FUNCTION_BLOCK "AutoSusDoor"	// FB 20
TITLE = pneum.RüstplTüren
//------------------------------------------------------------------------------
//version:      0.1 / 10.09.2007
//author:       H.Scheuenstuhl
//modification: Prototyp
//------------------------------------------------------------------------------
AUTHOR : SPAC_slh
FAMILY : AUTOMAT
NAME : SusDoor
VERSION : 0.1
VAR_INPUT
  iMode : BYTE ;	//Funktion:
  iSafetyEdgeMonitoringTim : BYTE ;	//Zeit Schaltleistenüberwachung (in 0.1 sek, BCD-codiert!)
  iOnly1SusDoor : BOOL ;	//einflügelige Rüstplatztür (links)
  iAutoReverse : BOOL ;	//0: sofort.Abschalten  1: Reversierbetrieb wenn Schaltleiste betätigt
END_VAR
VAR
  fk : ARRAY  [0 .. 15 ] OF //Flankenhilfsmerker [n]
  BOOL ;
  hvFEin : BOOL ;	//Hauptventil Fehler:Einschaltüberwachung
  hvFUnt : BOOL ;	//Hauptventil Fehler:Unterbrechungsüberwachung
  LBewTzu : BOOL ;	//letzte Bewegung:Türen schliessen
  SafetyEdgeActuated : BOOL ;	//Schaltleiste betätigt (wenn Türe(n) nicht geschlossen)
  SafetyEdgeReverseMove : BOOL ;	//Schaltleiste betätigt: Türen Rücklauf = Öffnen (Reversierung)
  SafetyEdgePressureOff : BOOL ;	//Schaltleiste betätigt: Pneumatik Druck aus
  SfCloseDoor : BOOL ;	//Schritt fertig:Tür schliessen
  SfOpenDoor : BOOL ;	//Schritt fertig:Tür öffnen
  oeffnFEin : BOOL ;	//Drucküberwachung RpTüren öffnen Fehler:Einschaltüberwachung
  oeffnFUnt : BOOL ;	//Drucküberwachung RpTüren öffnen Fehler:Unterbrechungsüberwachung
  schlFEin : BOOL ;	//Drucküberwachung RpTüren schliessen Fehler:Einschaltüberwachung
  schlFUnt : BOOL ;	//Drucküberwachung RpTüren schliessen Fehler:Unterbrechungsüberwachung
  Luftvh : BOOL ;	//Druckluft für Antrieb der Rüstplatztüren vorhanden
  LockManualOperate : BOOL ;	//Tastensperre nach Fehlbedienung
  SrCloseDoor : BOOL ;	//Schritt:Türen schliessen
  SrOpenDoor : BOOL ;	//Schritt:Türen öffnen
END_VAR
VAR_TEMP
  svAr1 : DWORD ;
  WertInt : INT ;	//Wert integer
  SLUeZeit : S5TIME ;	//s5-Zeitwert Schaltleistenüberwachung
  Mod : ARRAY  [0 .. 15 ] OF //Modus dekodiert, 1 aus 16
  BOOL ;
  LOp0 : BOOL ;	//lokaler Operationsmerker 0, Zwischenmerker
  LOp1 : BOOL ;	//lokaler Operationsmerker 1, Zwischenmerker
  Fa : BOOL ;	//Freigabe Ausgänge
  SusDoorAutoOpen : BOOL ;	//Modus: Rüstplatztür automatisch öffnen nach Palettenwechsel
  AutoEnablePc : BOOL ;	//Modus:automatisches Setzen der PW-Freigabe nach Rüstplatztür zu
  SusDoorOpened : BOOL ;	//Rüstlatztüren sind vollständig geöffnet
  ModeSusDoorAdjust : BOOL ;	//Rüstplatztüren: Betriebsart Einrichten
  ModeSusDoorAuto : BOOL ;	//Rüstplatztüren: Betriebsart Automatik
  AnfTzu1 : BOOL ;	//Anforderung Türen schliessen
  AnfTauf1 : BOOL ;	//Anforderung Türen öffnen
  MachineOn : BOOL ;	//Maschine ist ein
  afbTzu : BOOL ;	//Türen schliessen ausführbar
  afbTauf : BOOL ;	//Türen öffnen ausführbar
  SusDoorFault : BOOL ;	//Sammelsignal: Rüstplatztür(en) gestört
  CloseManual : BOOL ;	//Taster: Türen schliessen
  OpenManual : BOOL ;	//Taster: Türen öffnen
  CloseByRobot : BOOL ;	//Werkstücklader: Türen schliessen
  OpenByRobot : BOOL ;	//Werkstücklader: Türen öffnen
END_VAR
BEGIN
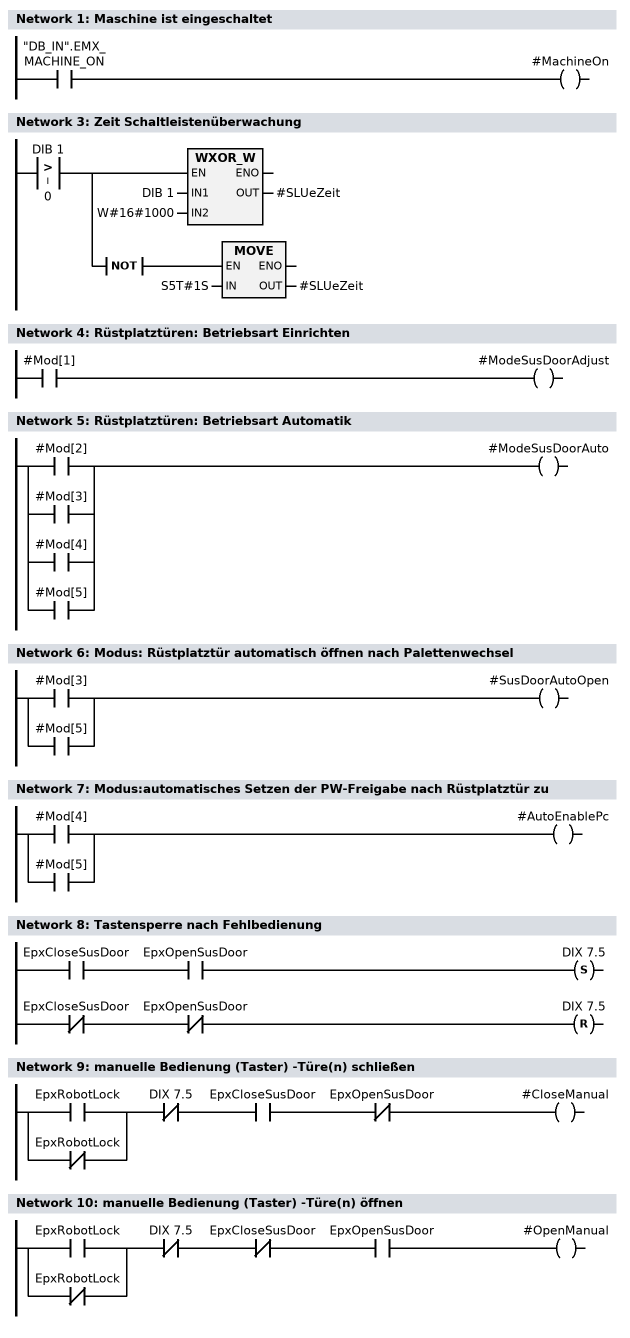
NETWORK
TITLE = Maschine ist eingeschaltet
      A     "DB_IN".EMX_MACHINE_ON;
      =     #MachineOn;
NETWORK
TITLE = iModus dekodieren
//Modus_1: Handbetrieb, Einrichtbetrieb, Tippbetrieb
//Modus_2: Tippen fährt bis Endlage erreicht
//Modus_3: Tippen fährt bis Endlage erreicht
//         nach PW fährt Türe automatisch auf
//Modus_4: Tippen fährt bis Endlage erreicht
//         nach Schließen wird PW-Freigabe gesetzt
//Modus_5: Tippen fährt bis Endlage erreicht
//         nach PW fährt Türe automatisch auf
//         nach Schließen wird PW-Freigabe gesetzt
      L     DIB 0;
      AW    W#16#F;	//Begrenzung auf 0..15, dadurch keine weitere Prüfung erforderlich
      TAR1  #svAr1;
      LAR1  P##Mod;
      L     B#16#0;
      T     LW [AR1,P#0.0];
      TAK;
      +AR1;
      A     "M_HIGH";
      S     L [AR1,P#0.0];
      LAR1  #svAr1;
NETWORK
TITLE = Zeit Schaltleistenüberwachung
//Zuordnung der Zeit (über Konstante S5T); Dekadenbyte = 1 ==> 0,1sec
      L     DIB 1;
      L     0;
      >I;
      =     L 13.0;
      A     L 13.0;
      JNB   _001;
      L     DIB 1;
      L     W#16#1000;
      XOW;
      T     #SLUeZeit;
_001: NOP   0;
      A     L 13.0;
      NOT;
      JNB   _002;
      L     S5T#1S;
      T     #SLUeZeit;
_002: NOP   0;
NETWORK
TITLE = Rüstplatztüren: Betriebsart Einrichten
//Modus_1: Handbetrieb, Einrichtbetrieb, Tippbetrieb
      A     #Mod[1];
      =     #ModeSusDoorAdjust;
NETWORK
TITLE = Rüstplatztüren: Betriebsart Automatik
//Modus_2: Tippen fährt bis Endlage erreicht
//Modus_3: Tippen fährt bis Endlage erreicht
//         nach PW fährt Türe automatisch auf
//Modus_4: Tippen fährt bis Endlage erreicht
//         nach Schließen wird PW-Freigabe gesetzt
//Modus_5: Tippen fährt bis Endlage erreicht
//         nach PW fährt Türe automatisch auf
//         nach Schließen wird PW-Freigabe gesetzt
      O     #Mod[2];
      O     #Mod[3];
      O     #Mod[4];
      O     #Mod[5];
      =     #ModeSusDoorAuto;
NETWORK
TITLE = Modus: Rüstplatztür automatisch öffnen nach Palettenwechsel
//Modus_3: Tippen fährt bis Endlage erreicht
//         nach PW fährt Türe automatisch auf
//Modus_5: Tippen fährt bis Endlage erreicht
//         nach PW fährt Türe automatisch auf
//         nach Schließen wird PW-Freigabe gesetzt
      O     #Mod[3];
      O     #Mod[5];
      =     #SusDoorAutoOpen;
NETWORK
TITLE = Modus:automatisches Setzen der PW-Freigabe nach Rüstplatztür zu
//Modus_4: Tippen fährt bis Endlage erreicht
//         nach Schließen wird PW-Freigabe gesetzt
//Modus_5: Tippen fährt bis Endlage erreicht
//         nach PW fährt Türe automatisch auf
//         nach Schließen wird PW-Freigabe gesetzt
      O     #Mod[4];
      O     #Mod[5];
      =     #AutoEnablePc;
NETWORK
TITLE = Tastensperre nach Fehlbedienung
      A     "EpxCloseSusDoor";
      A     "EpxOpenSusDoor";
      S     DIX 7.5;
      AN    "EpxCloseSusDoor";
      AN    "EpxOpenSusDoor";
      R     DIX 7.5;
      NOP   0;
NETWORK
TITLE = manuelle Bedienung (Taster) -Türe(n) schließen
      A(;
      O     "EpxRobotLock";
      ON    "EpxRobotLock";
      );
      AN    DIX 7.5;
      A     "EpxCloseSusDoor";
      AN    "EpxOpenSusDoor";
      =     #CloseManual;
NETWORK
TITLE = manuelle Bedienung (Taster) -Türe(n) öffnen
      A(;
      O     "EpxRobotLock";
      ON    "EpxRobotLock";
      );
      AN    DIX 7.5;
      AN    "EpxCloseSusDoor";
      A     "EpxOpenSusDoor";
      =     #OpenManual;
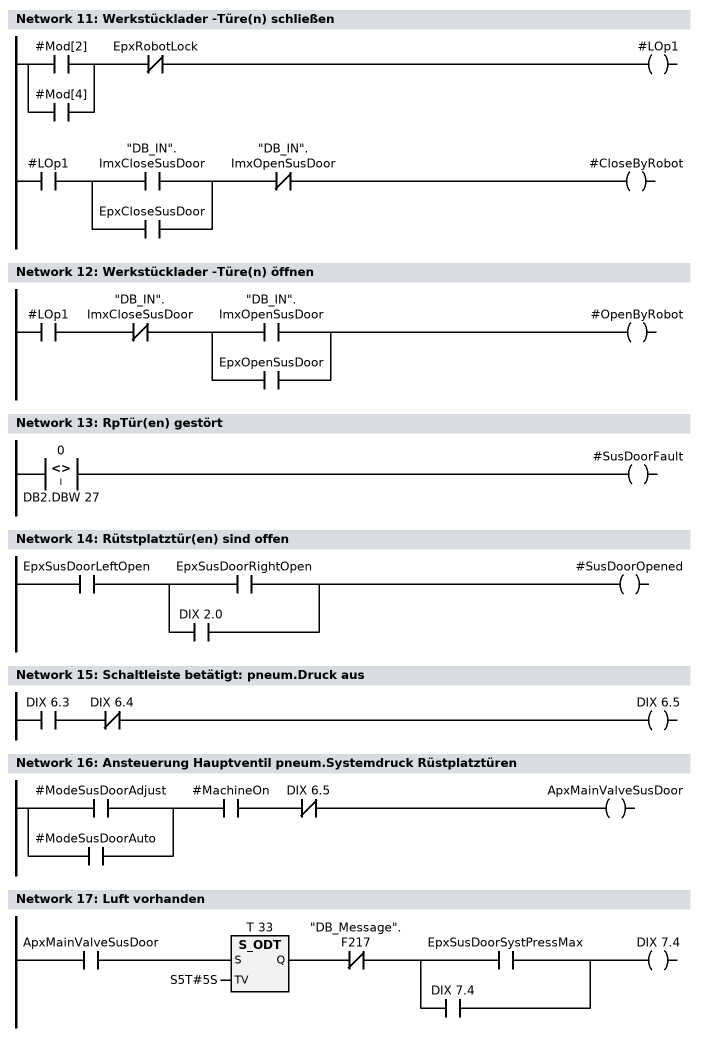
NETWORK
TITLE = Werkstücklader -Türe(n) schließen
//Modus_2: Tippen fährt bis Endlage erreicht
//Modus_4: Tippen fährt bis Endlage erreicht
//         nach Schließen wird PW-Freigabe gesetzt
      A(;
      O     #Mod[2];
      O     #Mod[4];
      );
      AN    "EpxRobotLock";
      =     #LOp1;
      A     #LOp1;
      A(;
      O     "DB_IN".ImxCloseSusDoor;
      O     "EpxCloseSusDoor";
      );
      AN    "DB_IN".ImxOpenSusDoor;
      =     #CloseByRobot;
NETWORK
TITLE = Werkstücklader -Türe(n) öffnen
      A     #LOp1;
      AN    "DB_IN".ImxCloseSusDoor;
      A(;
      O     "DB_IN".ImxOpenSusDoor;
      O     "EpxOpenSusDoor";
      );
      =     #OpenByRobot;
NETWORK
TITLE = RpTür(en) gestört
//DB2.DBW27 = Fehlermeldungen 217 bis 232
      L     0;
      L     DB2.DBW 27;
      <>I;
      =     #SusDoorFault;
NETWORK
TITLE = Rütstplatztür(en) sind offen
//Wenn nur eine Rüstplatztüre ausgewählt wird, dann ist die "rechte Türe" 
//gebrückt.
      A     "EpxSusDoorLeftOpen";
      A(;
      O     "EpxSusDoorRightOpen";
      O     DIX 2.0;
      );
      =     #SusDoorOpened;
NETWORK
TITLE = Schaltleiste betätigt: pneum.Druck aus
      A     DIX 6.3;
      AN    DIX 6.4;
      =     DIX 6.5;
NETWORK
TITLE = Ansteuerung Hauptventil pneum.Systemdruck Rüstplatztüren
      A(;
      O     #ModeSusDoorAdjust;
      O     #ModeSusDoorAuto;
      );
      A     #MachineOn;
      AN    DIX 6.5;
      =     "ApxMainValveSusDoor";
NETWORK
TITLE = Luft vorhanden
      A(;
      A     "ApxMainValveSusDoor";
      L     S5T#5S;
      SD    T 33;
      NOP   0;
      NOP   0;
      NOP   0;
      A     T 33;
      );
      AN    "DB_Message".F217;
      A(;
      O     "EpxSusDoorSystPressMax";
      O     DIX 7.4;
      );
      =     DIX 7.4;
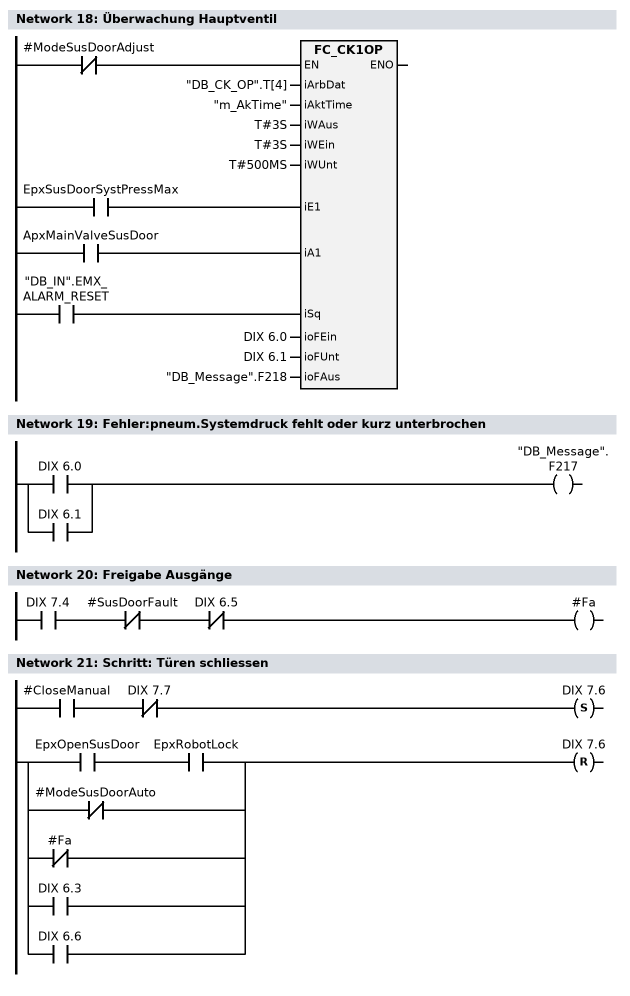
NETWORK
TITLE = Überwachung Hauptventil
      A     "EpxSusDoorSystPressMax";
      =     L 13.0;
      BLD   103;
      A     "ApxMainValveSusDoor";
      =     L 13.1;
      BLD   103;
      A     "DB_IN".EMX_ALARM_RESET;
      =     L 13.2;
      BLD   103;
      AN    #ModeSusDoorAdjust;
      JNB   _003;
      CALL  "FC_CK1OP" (
           iArbDat                  := "DB_CK_OP".T[4],
           iAktTime                 := "m_AkTime",
           iWAus                    := T#3S,
           iWEin                    := T#3S,
           iWUnt                    := T#500MS,
           iE1                      := L 13.0,
           iA1                      := L 13.1,
           iSq                      := L 13.2,
           ioFEin                   := DIX 6.0,
           ioFUnt                   := DIX 6.1,
           ioFAus                   := "DB_Message".F218);
_003: NOP   0;
NETWORK
TITLE = Fehler:pneum.Systemdruck fehlt oder kurz unterbrochen
      O     DIX 6.0;
      O     DIX 6.1;
      =     "DB_Message".F217;
NETWORK
TITLE = Freigabe Ausgänge
      A     DIX 7.4;
      AN    #SusDoorFault;
      AN    DIX 6.5;
      =     #Fa;
NETWORK
TITLE = Schritt: Türen schliessen
      A     #CloseManual;
      AN    DIX 7.7;
      S     DIX 7.6;
      A(;
      A     "EpxOpenSusDoor";
      A     "EpxRobotLock";
      ON    #ModeSusDoorAuto;
      ON    #Fa;
      O     DIX 6.3;
      O     DIX 6.6;
      );
      R     DIX 7.6;
      NOP   0;
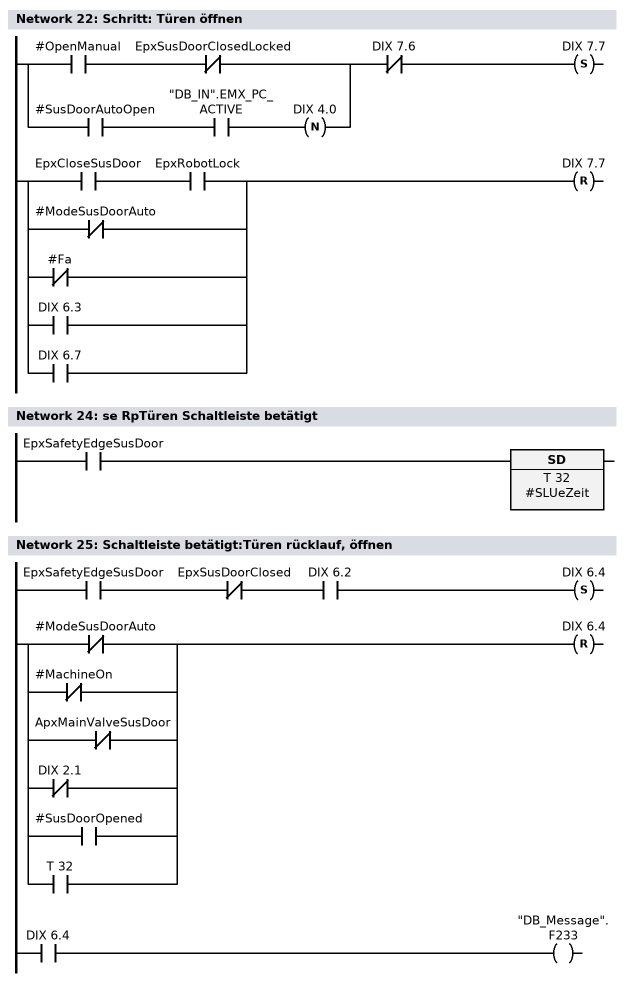
NETWORK
TITLE = Schritt: Türen öffnen
      A(;
      A     #OpenManual;
      AN    "EpxSusDoorClosedLocked";
      O(;
      A     #SusDoorAutoOpen;
      A     "DB_IN".EMX_PC_ACTIVE;
      FN    DIX 4.0;
      );
      );
      AN    DIX 7.6;
      S     DIX 7.7;
      A(;
      A     "EpxCloseSusDoor";
      A     "EpxRobotLock";
      ON    #ModeSusDoorAuto;
      ON    #Fa;
      O     DIX 6.3;
      O     DIX 6.7;
      );
      R     DIX 7.7;
      NOP   0;
NETWORK
TITLE = Schaltleiste an Rüstplatztüren betätigt
      A(;
      A     "DB_IN".EMX_ALARM_RESET;
      R     DIX 6.3;
      A     "EpxSafetyEdgeSusDoor";
      AN    "EpxSusDoorClosed";
      S     DIX 6.3;
      A     DIX 6.3;
      );
      AN    "DB_Message".F233;
      =     "DB_Message".F234;
NETWORK
TITLE = se RpTüren Schaltleiste betätigt
      A     "EpxSafetyEdgeSusDoor";
      L     #SLUeZeit;
      SD    T 32;
NETWORK
TITLE = Schaltleiste betätigt:Türen rücklauf, öffnen
      A     "EpxSafetyEdgeSusDoor";
      AN    "EpxSusDoorClosed";
      A     DIX 6.2;
      S     DIX 6.4;
      A(;
      ON    #ModeSusDoorAuto;
      ON    #MachineOn;
      ON    "ApxMainValveSusDoor";
      ON    DIX 2.1;
      O     #SusDoorOpened;
      O     T 32;
      );
      R     DIX 6.4;
      A     DIX 6.4;
      =     "DB_Message".F233;
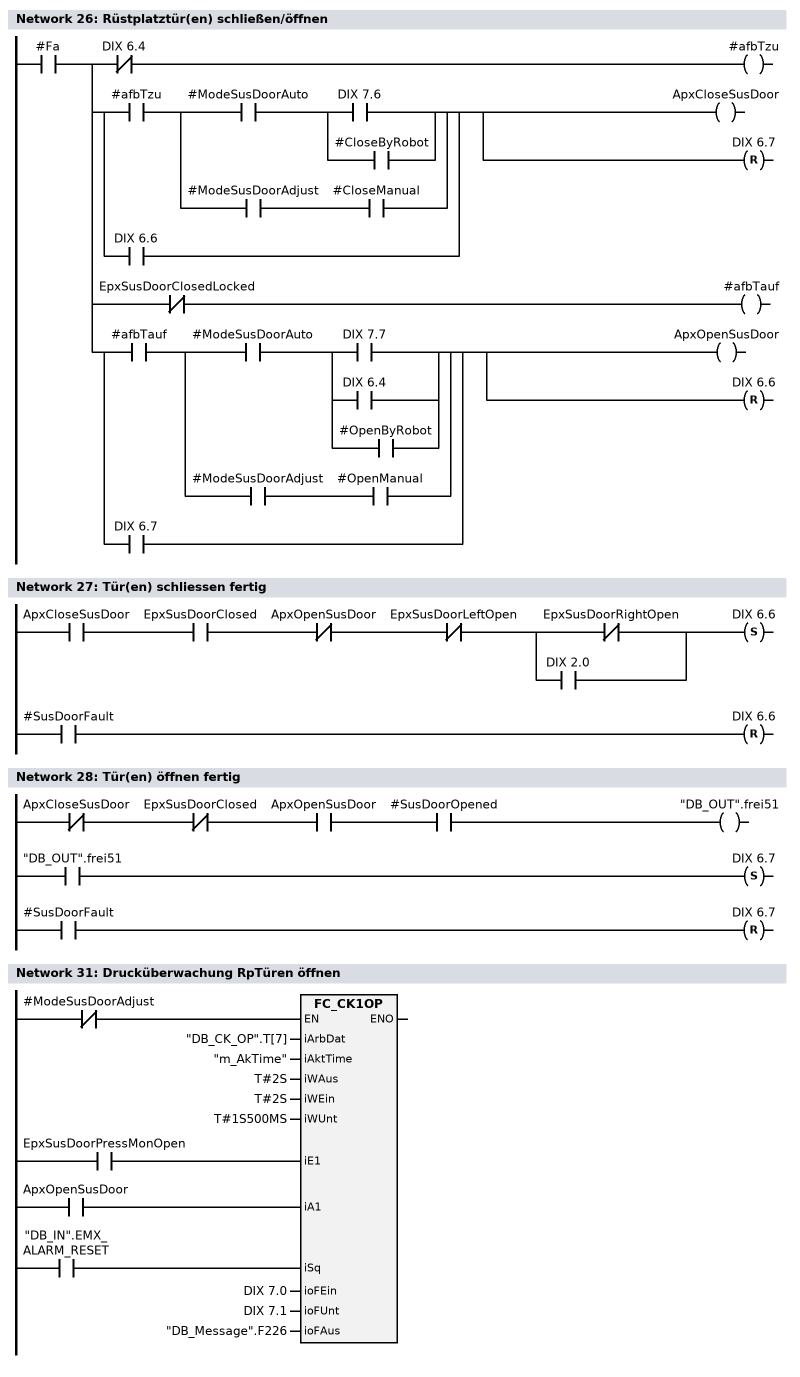
NETWORK
TITLE = Rüstplatztür(en) schließen/öffnen
      A     #Fa;
      =     L 13.0;
      A     L 13.0;
      AN    DIX 6.4;
      =     #afbTzu;
      A     L 13.0;
      A(;
      A     #afbTzu;
      A(;
      A     #ModeSusDoorAuto;
      A(;
      O     DIX 7.6;
      O     #CloseByRobot;
      );
      O;
      A     #ModeSusDoorAdjust;
      A     #CloseManual;
      );
      O     DIX 6.6;
      );
      =     "ApxCloseSusDoor";
      R     DIX 6.7;
      A     L 13.0;
      AN    "EpxSusDoorClosedLocked";
      =     #afbTauf;
      A     L 13.0;
      A(;
      A     #afbTauf;
      A(;
      A     #ModeSusDoorAuto;
      A(;
      O     DIX 7.7;
      O     DIX 6.4;
      O     #OpenByRobot;
      );
      O;
      A     #ModeSusDoorAdjust;
      A     #OpenManual;
      );
      O     DIX 6.7;
      );
      =     "ApxOpenSusDoor";
      R     DIX 6.6;
NETWORK
TITLE = Tür(en) schliessen fertig
      A     "ApxCloseSusDoor";
      A     "EpxSusDoorClosed";
      AN    "ApxOpenSusDoor";
      AN    "EpxSusDoorLeftOpen";
      A(;
      ON    "EpxSusDoorRightOpen";
      O     DIX 2.0;
      );
      S     DIX 6.6;
      A     #SusDoorFault;
      R     DIX 6.6;
      NOP   0;
NETWORK
TITLE = Tür(en) öffnen fertig
      AN    "ApxCloseSusDoor";
      AN    "EpxSusDoorClosed";
      A     "ApxOpenSusDoor";
      A     #SusDoorOpened;
      =     "DB_OUT".frei51;
      A     "DB_OUT".frei51;
      S     DIX 6.7;
      A     #SusDoorFault;
      R     DIX 6.7;
      NOP   0;
NETWORK
TITLE = Endschalterüberwachung RpTür links
      A     "EpxSusDoorLeftOpen";
      =     L 13.0;
      BLD   103;
      A     "ApxOpenSusDoor";
      =     L 13.1;
      BLD   103;
      A     "EpxSusDoorClosed";
      =     L 13.2;
      BLD   103;
      A     "ApxCloseSusDoor";
      =     L 13.3;
      BLD   103;
      A     "M_LOW";
      =     L 13.4;
      BLD   103;
      A     "DB_IN".EMX_ALARM_RESET;
      =     L 13.5;
      BLD   103;
      A     "M_LOW";
      =     L 13.6;
      BLD   103;
      A     "M_LOW";
      =     L 13.7;
      BLD   103;
      A     "M_LOW";
      =     L 14.0;
      BLD   103;
      AN    #ModeSusDoorAdjust;
      JNB   _004;
      BLD   1;
      L     W#16#1002;
      T     LW 15;
      L     14;
      T     LW 17;
      L     101;
      T     LW 19;
      L     P#DBX 70.0;
      T     LD 21;
      L     L#100;
      T     LD 25;
      L     L#7000;
      T     LD 29;
      L     L#1000;
      T     LD 33;
      A     "DB_Message".Me737;
      =     L 37.0;
      A     "DB_Message".Me738;
      =     L 37.1;
      A     "DB_Message".F219;
      =     L 37.2;
      A     "DB_Message".F220;
      =     L 37.3;
      A     "DB_Message".F221;
      =     L 37.4;
      UC    "FC_CK2OP";
      {     P#L 15.0, P#M 12.0, P#L 25.0, P#L 29.0, P#L 33.0, P#L 13.0, P#L 13.1, P#L 13.2, P#L 13.3, P#L 13.4, P#L 13.5, P#L 13.6, P#L 13.7, P#L 14.0, P#L 37.0, P#L 37.1, P#L 37.2, P#L 37.3, P#L 37.4 };
      A     L 37.0;
      =     "DB_Message".Me737;
      A     L 37.1;
      =     "DB_Message".Me738;
      A     L 37.2;
      =     "DB_Message".F219;
      A     L 37.3;
      =     "DB_Message".F220;
      A     L 37.4;
      =     "DB_Message".F221;
      BLD   2;
_004: NOP   0;
NETWORK
TITLE = Endschalterüberwachung RpTür rechts
      A     "EpxSusDoorRightOpen";
      =     L 13.0;
      BLD   103;
      A     "ApxOpenSusDoor";
      =     L 13.1;
      BLD   103;
      A     "EpxSusDoorClosed";
      =     L 13.2;
      BLD   103;
      A     "ApxCloseSusDoor";
      =     L 13.3;
      BLD   103;
      A     "M_LOW";
      =     L 13.4;
      BLD   103;
      A     "DB_IN".EMX_ALARM_RESET;
      =     L 13.5;
      BLD   103;
      A     "M_LOW";
      =     L 13.6;
      BLD   103;
      A     "M_LOW";
      =     L 13.7;
      BLD   103;
      A     "M_LOW";
      =     L 14.0;
      BLD   103;
      AN    #ModeSusDoorAdjust;
      AN    DIX 2.0;
      JNB   _005;
      BLD   1;
      L     W#16#1002;
      T     LW 15;
      L     14;
      T     LW 17;
      L     101;
      T     LW 19;
      L     P#DBX 84.0;
      T     LD 21;
      L     L#100;
      T     LD 25;
      L     L#7000;
      T     LD 29;
      L     L#1000;
      T     LD 33;
      A     "DB_Message".Me739;
      =     L 37.0;
      A     "DB_Message".Me740;
      =     L 37.1;
      A     "DB_Message".F222;
      =     L 37.2;
      A     "DB_Message".F223;
      =     L 37.3;
      A     "DB_Message".F224;
      =     L 37.4;
      UC    "FC_CK2OP";
      {     P#L 15.0, P#M 12.0, P#L 25.0, P#L 29.0, P#L 33.0, P#L 13.0, P#L 13.1, P#L 13.2, P#L 13.3, P#L 13.4, P#L 13.5, P#L 13.6, P#L 13.7, P#L 14.0, P#L 37.0, P#L 37.1, P#L 37.2, P#L 37.3, P#L 37.4 };
      A     L 37.0;
      =     "DB_Message".Me739;
      A     L 37.1;
      =     "DB_Message".Me740;
      A     L 37.2;
      =     "DB_Message".F222;
      A     L 37.3;
      =     "DB_Message".F223;
      A     L 37.4;
      =     "DB_Message".F224;
      BLD   2;
_005: NOP   0;
NETWORK
TITLE = Drucküberwachung RpTüren öffnen
      A     "EpxSusDoorPressMonOpen";
      =     L 13.0;
      BLD   103;
      A     "ApxOpenSusDoor";
      =     L 13.1;
      BLD   103;
      A     "DB_IN".EMX_ALARM_RESET;
      =     L 13.2;
      BLD   103;
      AN    #ModeSusDoorAdjust;
      JNB   _006;
      CALL  "FC_CK1OP" (
           iArbDat                  := "DB_CK_OP".T[7],
           iAktTime                 := "m_AkTime",
           iWAus                    := T#2S,
           iWEin                    := T#2S,
           iWUnt                    := T#1S500MS,
           iE1                      := L 13.0,
           iA1                      := L 13.1,
           iSq                      := L 13.2,
           ioFEin                   := DIX 7.0,
           ioFUnt                   := DIX 7.1,
           ioFAus                   := "DB_Message".F226);
_006: NOP   0;
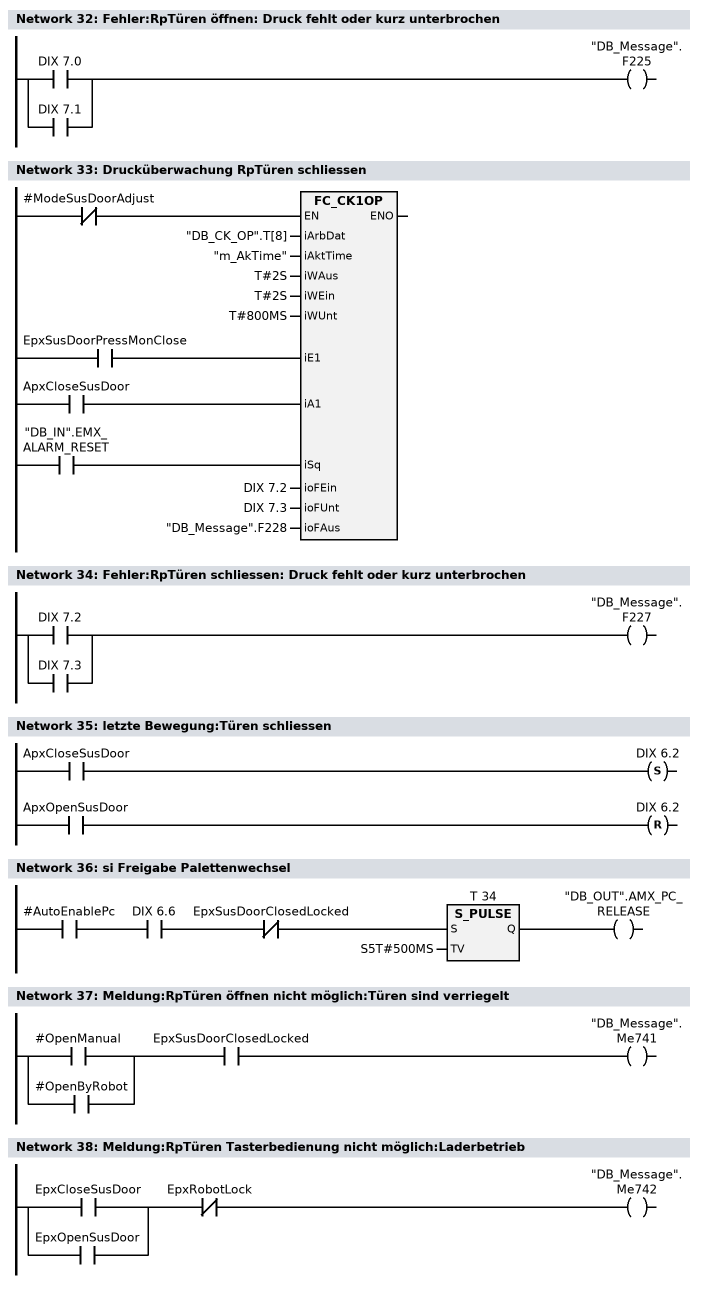
NETWORK
TITLE = Fehler:RpTüren öffnen: Druck fehlt oder kurz unterbrochen
      O     DIX 7.0;
      O     DIX 7.1;
      =     "DB_Message".F225;
NETWORK
TITLE = Drucküberwachung RpTüren schliessen
      A     "EpxSusDoorPressMonClose";
      =     L 13.0;
      BLD   103;
      A     "ApxCloseSusDoor";
      =     L 13.1;
      BLD   103;
      A     "DB_IN".EMX_ALARM_RESET;
      =     L 13.2;
      BLD   103;
      AN    #ModeSusDoorAdjust;
      JNB   _007;
      CALL  "FC_CK1OP" (
           iArbDat                  := "DB_CK_OP".T[8],
           iAktTime                 := "m_AkTime",
           iWAus                    := T#2S,
           iWEin                    := T#2S,
           iWUnt                    := T#800MS,
           iE1                      := L 13.0,
           iA1                      := L 13.1,
           iSq                      := L 13.2,
           ioFEin                   := DIX 7.2,
           ioFUnt                   := DIX 7.3,
           ioFAus                   := "DB_Message".F228);
_007: NOP   0;
NETWORK
TITLE = Fehler:RpTüren schliessen: Druck fehlt oder kurz unterbrochen
      O     DIX 7.2;
      O     DIX 7.3;
      =     "DB_Message".F227;
NETWORK
TITLE = letzte Bewegung:Türen schliessen
      A     "ApxCloseSusDoor";
      S     DIX 6.2;
      A     "ApxOpenSusDoor";
      R     DIX 6.2;
      NOP   0;
NETWORK
TITLE = si Freigabe Palettenwechsel
      A     #AutoEnablePc;
      A     DIX 6.6;
      AN    "EpxSusDoorClosedLocked";
      L     S5T#500MS;
      SP    T 34;
      NOP   0;
      NOP   0;
      NOP   0;
      A     T 34;
      =     "DB_OUT".AMX_PC_RELEASE;
NETWORK
TITLE = Meldung:RpTüren öffnen nicht möglich:Türen sind verriegelt
      A(;
      O     #OpenManual;
      O     #OpenByRobot;
      );
      A     "EpxSusDoorClosedLocked";
      =     "DB_Message".Me741;
NETWORK
TITLE = Meldung:RpTüren Tasterbedienung nicht möglich:Laderbetrieb
      A(;
      O     "EpxCloseSusDoor";
      O     "EpxOpenSusDoor";
      );
      AN    "EpxRobotLock";
      =     "DB_Message".Me742;
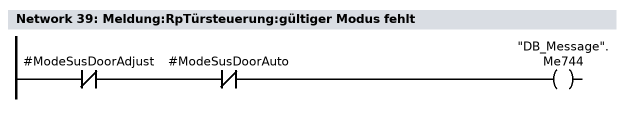
NETWORK
TITLE = Meldung:RpTürsteuerung:gültiger Modus fehlt
      AN    #ModeSusDoorAdjust;
      AN    #ModeSusDoorAuto;
      =     "DB_Message".Me744;
END_FUNCTION_BLOCK

FUNCTION_BLOCK "MESSAGE_OUT"	// FB 100
TITLE = Erfassung Alarm-/Betriebsmeldungen
//________________________________________________________________________________
//$Revision: x.y $
//$Date: 2005/04/26 0:0:0CET $
//$Author: slh $
//$ProjectRevision: Last Checkpoint: m.n $
//
//-------------------------------------------------------------------------------
//*COPYRIGHT BY SCHEUENSTUHL PAC - GERMANY
//*Softwareentwicklung
//erstellt: 27.04.2005; Helmut Scheuenstuhl (slh); Scheuenstuhl PAC
//Änderung: Datum / Abteilung / Name / Version x.y
//Änderung: 
//        :
//-------------------------------------------------------------------------------
//Beschreibung
//Der Baustein dient zur Nummerngenerierung von Fehler-/Betriebsmeldungen. Die
//vom Anwenderprg. erzeugten Alarme --- Alarm   001..512   -> DB2.DBX0.0-DBX63.7
//                 bzw. Meldungen ----- Meldung 513..1024  -> DB2.DBX64.0-DBX127.7
//werden mit der fest zugeordneten Nr. erfasst und am Ausgang oAlMldNr wie folgt
//ausgegeben:
//Bei mehreren anstehenden Alarmen/Meldungen werden in einem durch iZeitwert iVm. 
//iTimer festgelegten Zeitraster alle anstehenden Alarme/Meldungen auf oAlMldNr
//durchgeschaltet. Alarme werden höherprior behandelt: Nur wenn kein Alarm 
//ansteht werden Meldungen ausgegeben.
AUTHOR : SPAC_slh
NAME : MSG
VERSION : 0.1
VAR_INPUT
  IN_TIM_TOGGLE : TIMER ;	//Zeit für Anzeigeintervall
  IN_S5T_TOGGLE : S5TIME ;	//Zeitwert für Anzeigeintervall
END_VAR
VAR_OUTPUT
  OUT_INT_MESSAGENUMBER : INT ;	//Alarm-/Meldungsnr.
END_VAR
VAR
  MStack : ARRAY  [0 .. 255 ] OF //Stack für Alarme/Meldungen
  INT ;
  wrStck : INT ;	//Stackzeiger beim Schreiben
  rdStck : INT ;	//Stackzeiger beim Lesen
END_VAR
VAR_TEMP
  svAr1 : DWORD ;	//Rettregister von AR1
  loopctr : INT ;	//Schleifenzähler
  ALMldNr : INT ;	//Alarm-/Meldungsnr.
  PrfWrd : WORD ;	//zu prüfendes Wort
  Bitmaske : WORD ;	//Bitmaske
  Bitnr : BYTE ;	//Bitnr.des gesetzten Bits
  LOp1 : BOOL ;	//lokaler Operationsmerker 1, Zwischenmerker
END_VAR
BEGIN
NETWORK
TITLE = Initialisierung, Stack löschen
      OPN   "DB_Message";
      L     0;
      T     DIW 518;
      TAR1  #svAr1;
      LAR1  P##MStack;
      L     128;
cs01: L     0;
      T     DID [AR1,P#0.0];
      +AR1  P#4.0;
      TAK;
      LOOP  cs01;
NETWORK
TITLE = Erfassung Alarme
      L     0;
s011: T     #loopctr;
      SLW   4;	//slw3:Pointerformat slw1:Wortbreite
      LAR1;
      L     0;
      L     DBW [AR1,P#0.0];
      ==I;
      JC    m011;	//kein Alarmbit gesetzt, nächstes Wort prüfen
      CAW;	//Bytekorrektur
m014: T     #PrfWrd;
      DTR;
      SRD   23;	//im Exponent steht Bias und höchstes gesetztes Bit
      +     -127;	//Bias subtrahieren, bei 32Bit GleitpktZahlen sind das 127
      T     #Bitnr;
      L     #loopctr;
      SLW   4;	//Meldungsoffset pro Wort:hier 16
      +I;
      +     1;	//AlarmnrKorrektur:dbx0.0==Alarmnr.1
//---(1)--- Eintrag in AL-/Meldungspuffer ------------------
      LAR1  P##MStack;
      L     DIW 518;
      SLW   4;	//slw3:Pointerformat slw1:Wortbreite
      +AR1;
      TAK;
      T     DIW [AR1,P#0.0];
      L     255;
      L     DIW 518;
      >I;
      JCN   m013;
      +     1;
      T     DIW 518;
//---(1)----------------------------------------------------
m013: L     0;
      LAR1  P##Bitmaske;
      T     LW [AR1,P#0.0];	//clr Bitmaske
      L     #Bitnr;
      +AR1;
      S     L [AR1,P#0.0];
      L     #Bitmaske;
      CAW;	//Bytekorrektur
      INVI;
      L     #PrfWrd;
      AW;
      L     0;
      <>I;
      TAK;
      JC    m014;	//wenn weiteres Bit gesetzt ist, erneut prüfen
m011: L     31;
      L     #loopctr;
      +     1;
      >=I;
      JC    s011;
NETWORK
TITLE = Erfassung Meldungen
      L     0;
      L     DIW 6;
      <>I;
      JC    m029;	//Wenn schon Eintrag durch Alarme erfolgt, keine Meldungen mehr suchen
      L     32;
s021: T     #loopctr;
      SLW   4;	//slw3:Pointerformat slw1:Wortbreite
      LAR1;
      L     0;
      L     DBW [AR1,P#0.0];
      ==I;
      JC    m021;	//kein Alarmbit gesetzt, nächstes Wort prüfen
      CAW;	//Bytekorrektur
m024: T     #PrfWrd;
      DTR;
      SRD   23;	//im Exponent steht Bias und höchstes gesetztes Bit
      +     -127;	//Bias subtrahieren, bei 32Bit GleitpktZahlen sind das 127
      T     #Bitnr;
      L     #loopctr;
      SLW   4;	//Meldungsoffset pro Wort:hier 16
      +I;
      +     1;	//AlarmnrKorrektur:dbx0.0==Alarmnr.1
//---(1)--- Eintrag in AL-/Meldungspuffer ------------------
      LAR1  P##MStack;
      L     DIW 518;
      SLW   4;	//slw3:Pointerformat slw1:Wortbreite
      +AR1;
      TAK;
      T     DIW [AR1,P#0.0];
      L     255;
      L     DIW 518;
      >I;
      JCN   m023;
      +     1;
      T     DIW 518;
//---(1)----------------------------------------------------
m023: L     0;
      LAR1  P##Bitmaske;
      T     LW [AR1,P#0.0];	//clr Bitmaske
      L     #Bitnr;
      +AR1;
      S     L [AR1,P#0.0];
      L     #Bitmaske;
      CAW;	//Bytekorrektur
      INVI;
      L     #PrfWrd;
      AW;
      L     0;
      <>I;
      TAK;
      JC    m024;	//wenn weiteres Bit gesetzt ist, erneut prüfen
m021: L     63;
      L     #loopctr;
      +     1;
      >=I;
      JC    s021;
m029: NOP   0;
NETWORK
TITLE = Steuerung Stacklesezeiger
      LAR1  #svAr1;
      L     0;
      L     DIW 6;
      <>I;
      L     DIW 2;
      SD    T [DIW 0];
      JC    m044;
      L     0;
      T     DIW 520;	//rdStck auf Wert 0 setzen wenn keine Meldung ansteht
m044: AN    T [DIW 0];
      JC    m041;
      L     255;
      L     DIW 520;
      +     1;
      <I;
      JCN   m042;
      L     0;
m042: T     DIW 520;
      TAR1  #svAr1;
      LAR1  P##MStack;
      L     DIW 520;
      SLW   4;	//slw3:Pointerformat slw1:Wortbreite
      +AR1;
      L     0;
      L     DIW [AR1,P#0.0];
      ==I;
      LAR1  #svAr1;
      JCN   m043;
      L     0;
      T     DIW 520;	//rdStck auf Wert 0 setzen wenn nächster Platz leer ist
m043: CLR;
      L     DIW 2;
      SD    T [DIW 0];
      SET;
      SD    T [DIW 0];
m041: TAR1  #svAr1;
      LAR1  P##MStack;
      L     DIW 520;
      SLW   4;	//slw3:Pointerformat slw1:Wortbreite
      +AR1;
      L     DIW [AR1,P#0.0];
      LAR1  #svAr1;
      T     #ALMldNr;
NETWORK
TITLE = Alarm-/Meldungsnr. zur Ausgabe
      L     #ALMldNr;
      T     DIW 4;
END_FUNCTION_BLOCK

FUNCTION "FUNCTIONS" : VOID	// FC 90
TITLE = Auswertung eines Datenwortes
//------------------------------------------------------------------------------
//version:      1.0 / 21.06.2007
//author:       H.Scheuenstuhl
//modification: Prototyp
//------------------------------------------------------------------------------
AUTHOR : APetz
FAMILY : GENERAL
NAME : General
VERSION : 1.0
VAR_INPUT
  iMaPar : WORD ;	//auszuwertender Maschinenparameter (BCD-Code)
  iDekade : BYTE ;	//mit welcher Dekade wird verglichen (0-3) für 10e0=Einer bis 10e3=Tausender
  iVglWert : BYTE ;	//Angabe des Wertes, mit dem verglichen werden soll
END_VAR
VAR_OUTPUT
  oMsb : BYTE ;	//höherwertiges Byte von iMaPar
  oLsb : BYTE ;	//niederwertiges Byte von iMaPar
  o10e0 : BYTE ;	//10e0-Dekade von iMaPar
  o10e1 : BYTE ;	//10e1-Dekade von iMaPar
  o10e2 : BYTE ;	//10e2-Dekade von iMaPar
  o10e3 : BYTE ;	//10e3-Dekade von iMaPar
  oVglTrue : BOOL ;	//log.1: iVglWert==iMaPar[Dekade]
END_VAR
VAR_TEMP
  MaParBcd : WORD ;
END_VAR
BEGIN
NETWORK
TITLE =
      L     #iMaPar;
      DTB;
      T     #MaParBcd;
      AW    W#16#F;
      T     #o10e0;
      L     #MaParBcd;
      AW    W#16#F0;
      SRW   4;
      T     #o10e1;
      L     #MaParBcd;
      AW    W#16#F00;
      SRW   8;
      T     #o10e2;
      L     #MaParBcd;
      AW    W#16#F000;
      SRW   12;
      T     #o10e3;
      L     #MaParBcd;
      AW    W#16#FF;
      BTI;
      T     #oLsb;
      L     #MaParBcd;
      CAW;
      AW    W#16#FF;
      BTI;
      T     #oMsb;
      L     #iDekade;
      JL    maxd;
      JU    m2e0;
      JU    m2e1;
      JU    m2e2;
      JU    m2e3;
maxd: CLR;
      JU    m002;
m2e0: L     #o10e0;
      JU    m001;
m2e1: L     #o10e1;
      JU    m001;
m2e2: L     #o10e2;
      JU    m001;
m2e3: L     #o10e3;
m001: L     #iVglWert;
      ==I;
m002: =     #oVglTrue;
END_FUNCTION

FUNCTION "CHANGE_BYTE" : VOID	// FC 91
//FUNKTION 1:
//
AUTHOR : A.Petz
VERSION : 0.1
VAR_INPUT
  I_ID : INT ;	//Identifikation der Funktion (Integer)
  W_MP : WORD ;	//Wert des Maschinenparameters
END_VAR
VAR_OUTPUT
  W_CHANGE_MP : WORD ;	//Wert des Maschinenparameters (angepasst an Reihenfolge der Bytes)
END_VAR
BEGIN
NETWORK
TITLE =
//Kehrt die Reihenfolge der Bytes in AKKU1-L
//Das Ergebnis wird in AKKU1-L gespeichert
//EN-Eingang gesetzt (bei KOP/FUP)?
//      U     BIE
//      SPBN  END1
      L     #I_ID;
      L     1;
      ==I;
      JCN   N_E1;
      L     #W_MP;
      CAW;
      T     #W_CHANGE_MP;
N_E1: NOP   0;
//Funktion wurde korrekt ausgeführt
//setzt ENO auf High
      SET;
      SAVE;
END_FUNCTION

FUNCTION "SIGNAL" : VOID	// FC 92
TITLE = ALLGEMEINE SIGNALVERKNÜPFUNGEN
//Funktionen zum Bilden von diversen Signalverknüpfungen, die für 
//unterschiedliche Anwendungen verwendet werden können (z.B. 
//Betriebsdatenerfassung, Signalleuchte, ...)
AUTHOR : A.Petz
VERSION : 0.1
VAR_INPUT
  IN_INT_IDENTIFICATION : INT ;	//Funktionskennung der Signalverküpfung
END_VAR
VAR_OUTPUT
  OUT_BIT_SIGNAL : BOOL ;	//Ergebnis der Signalverknüpfung
END_VAR
VAR_TEMP
  TMP_INT_IDENTIFICATION : INT ;	//Identifiaktionsnummer der Funktion
  TMP_BIT_ENABLE : BOOL ;	//Bausteinfreigabe - Sammelstörung
END_VAR
BEGIN
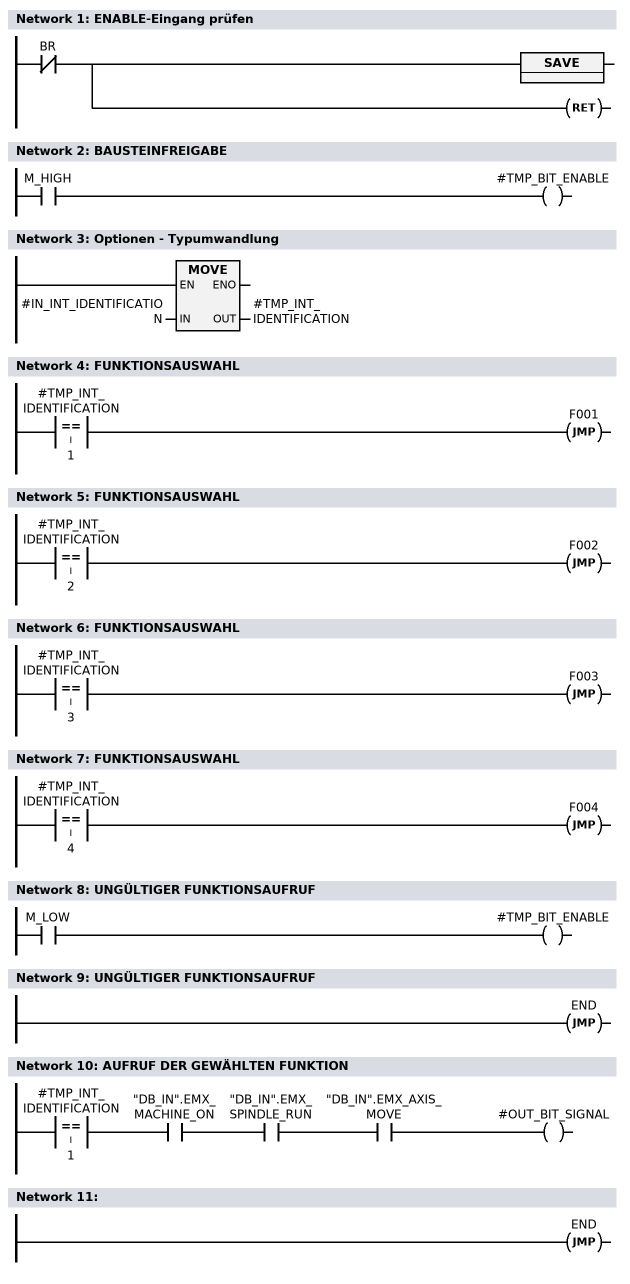
NETWORK
TITLE = ENABLE-Eingang prüfen
//Auswerten des BIE-Statusbit. Dieses entspricht dem EN (ENABLE)-Einganges bei 
//KOP/FUP. Wenn EN=FALSE dann verlasse Baustein.
      AN    BR;
      SAVE;
      BEC;
NETWORK
TITLE = BAUSTEINFREIGABE
//Fehlerauswertung Baustein intern:
//Bausteinfreigabe wird gesetzt
      A     "M_HIGH";
      =     #TMP_BIT_ENABLE;
NETWORK
TITLE = Optionen - Typumwandlung
//Konvertierung des "Identifikationsbytes" nach Integer
      L     #IN_INT_IDENTIFICATION;
      T     #TMP_INT_IDENTIFICATION;
      NOP   0;
NETWORK
TITLE = FUNKTIONSAUSWAHL
//Funktion mit Identifikation = 1 aufrufen
//Spindel läuft und mindestens eine Achse in Bewegung
//... wird bei "Not-Aus" zurückgesetzt.
      L     #TMP_INT_IDENTIFICATION;
      L     1;
      ==I;
      JC    F001;
NETWORK
TITLE = FUNKTIONSAUSWAHL
//Funktion mit Identifikation = 2 aufrufen
//Betriebsart MDA (Teach-In), SINGLE oder Betriebsart AUTOMATIK angewählt und 
//Programm läuft.
//... wird bei "Not-Aus" zurückgesetzt.
      L     #TMP_INT_IDENTIFICATION;
      L     2;
      ==I;
      JC    F002;
NETWORK
TITLE = FUNKTIONSAUSWAHL
//Funktion mit Identifikation = 3 aufrufen
//Maschine Ein und Betriebsart MANUAL angewählt.
      L     #TMP_INT_IDENTIFICATION;
      L     3;
      ==I;
      JC    F003;
NETWORK
TITLE = FUNKTIONSAUSWAHL
//Funktion mit Identifikation = 4 aufrufen
//Maschinenstörung (Fehlermeldung) oder Programm Ende oder Not-Aus
      L     #TMP_INT_IDENTIFICATION;
      L     4;
      ==I;
      JC    F004;
NETWORK
TITLE = UNGÜLTIGER FUNKTIONSAUFRUF
//Wenn keine gültige Identifikationsnummer übergeben wurde, wird das 
//Bausteinfreigabe (Sammelstörmeldung-Baustein) zurückgesetzt.
      A     "M_LOW";
      =     #TMP_BIT_ENABLE;
NETWORK
TITLE = UNGÜLTIGER FUNKTIONSAUFRUF
//Wenn keine gültige Identifikationsnummer übergeben wurde, wird an das 
//Programm-Ende gesprungen.
      JU    END;
NETWORK
TITLE = AUFRUF DER GEWÄHLTEN FUNKTION
//IDENTIFICATION = 1
//Spindel läuft und mindestens eine Achse in Bewegung
//... wird bei "Not-Aus" zurückgesetzt.
F001: A(;
      L     #TMP_INT_IDENTIFICATION;
      L     1;
      ==I;
      );
      A     "DB_IN".EMX_MACHINE_ON;
      A     "DB_IN".EMX_SPINDLE_RUN;
      A     "DB_IN".EMX_AXIS_MOVE;
      =     #OUT_BIT_SIGNAL;
NETWORK
TITLE =
      JU    END;	//      BEA   
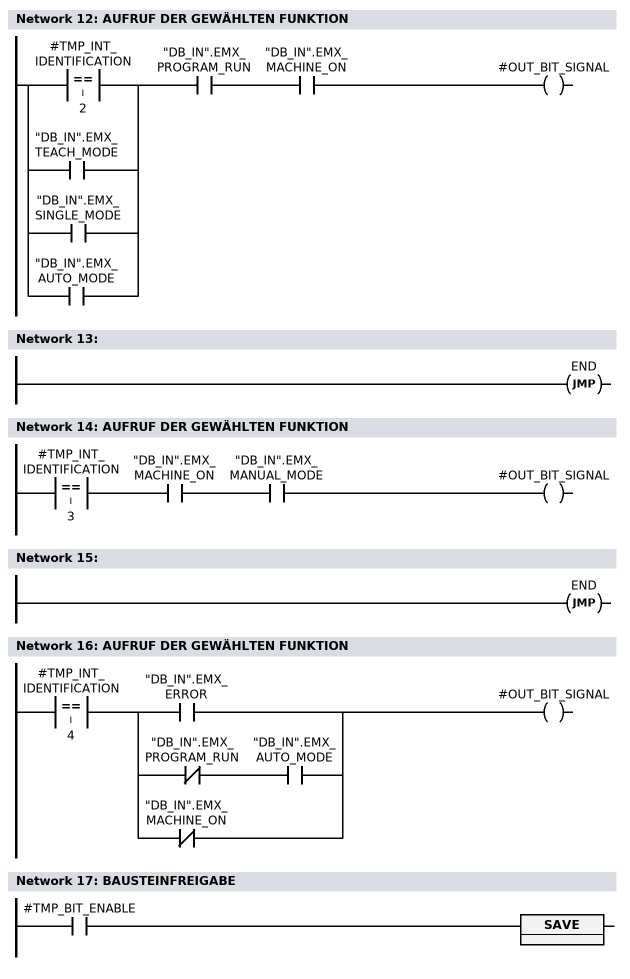
NETWORK
TITLE = AUFRUF DER GEWÄHLTEN FUNKTION
//IDENTIFICATION = 2
//Betriebsart MDA (Teach-In), SINGLE oder Betriebsart AUTOMATIK angewählt und 
//Programm läuft.
//... wird bei "Not-Aus" zurückgesetzt.
F002: A(;
      O(;
      L     #TMP_INT_IDENTIFICATION;
      L     2;
      ==I;
      );
      O     "DB_IN".EMX_TEACH_MODE;
      O     "DB_IN".EMX_SINGLE_MODE;
      O     "DB_IN".EMX_AUTO_MODE;
      );
      A     "DB_IN".EMX_PROGRAM_RUN;
      A     "DB_IN".EMX_MACHINE_ON;
      =     #OUT_BIT_SIGNAL;
NETWORK
TITLE =
      JU    END;	//      BEA   
NETWORK
TITLE = AUFRUF DER GEWÄHLTEN FUNKTION
//IDENTIFICATION = 3
//Maschine Ein und Betriebsart MANUAL angewählt.
F003: A(;
      L     #TMP_INT_IDENTIFICATION;
      L     3;
      ==I;
      );
      A     "DB_IN".EMX_MACHINE_ON;
      A     "DB_IN".EMX_MANUAL_MODE;
      =     #OUT_BIT_SIGNAL;
NETWORK
TITLE =
      JU    END;	//      BEA   
NETWORK
TITLE = AUFRUF DER GEWÄHLTEN FUNKTION
//IDENTIFICATION = 4
//Maschinenstörung (Fehlermeldung) oder Programm Ende (in Betriebsart 
//"Automatik") oder Not-Aus
F004: A(;
      L     #TMP_INT_IDENTIFICATION;
      L     4;
      ==I;
      );
      A(;
      O     "DB_IN".EMX_ERROR;
      O;
      AN    "DB_IN".EMX_PROGRAM_RUN;
      A     "DB_IN".EMX_AUTO_MODE;
      ON    "DB_IN".EMX_MACHINE_ON;
      );
      =     #OUT_BIT_SIGNAL;
NETWORK
TITLE = BAUSTEINFREIGABE
//Statusbit BIE=ENO setzen, wenn Funktion ohne Fehler durchlaufen wurde.
END:  A     #TMP_BIT_ENABLE;
      SAVE;
END_FUNCTION

FUNCTION "SELECT_TIME" : VOID	// FC 93
AUTHOR : A.Petz
VERSION : 0.2
VAR_INPUT
  iMdWert : WORD ;	//Wert des Maschinenparameters
  iMsb : BOOL ;	//Auswahl höherwertiges Byte des MdWertes (also Bits 8-15)
END_VAR
VAR_OUTPUT
  oWEin : TIME ;	//Wert für Einschaltverzögerung
  oWAus : TIME ;	//Wert für Auschaltverzögerung
END_VAR
VAR_TEMP
  WertBcd : WORD ;
END_VAR
BEGIN
NETWORK
TITLE = Typumwandlung
//Umwandlung des Eingangswortes in BCD-Code
      L     #iMdWert;
      DTB;
      T     #WertBcd;
NETWORK
TITLE = Auswertung niederwertiges Byte
      A     #iMsb;
      JC    e001;
      L     #WertBcd;
      AW    W#16#FF;
      L     0;
      ==I;
      JC    m010;
      L     #WertBcd;
      AW    W#16#F;
      +     3;
      L     1000;
      *I;
      T     #oWEin;
      L     #WertBcd;
      SRW   4;
      AW    W#16#F;
      SLW   2;
      +     2;
      L     1000;
      *I;
      T     #oWAus;
      JU    e001;
m010: L     T#10M;
      T     #oWEin;
      T     #oWAus;
e001: NOP   0;
NETWORK
TITLE = Auswertung höherwertiges Byte
      AN    #iMsb;
      JC    e002;
      L     #WertBcd;
      CAW;
      AW    W#16#FF;
      L     0;
      ==I;
      JC    m020;
      TAK;
      AW    W#16#F;
      +     3;
      L     1000;
      *I;
      T     #oWEin;
      L     #WertBcd;
      SRW   12;
      AW    W#16#F;
      SLW   2;
      +     2;
      L     1000;
      *I;
      T     #oWAus;
      JU    e002;
m020: L     T#10M;
      T     #oWEin;
      T     #oWAus;
e002: NOP   0;
END_FUNCTION

FUNCTION "MachineType" : VOID	// FC 94
//------------------------------------------------------------------------------
//version:      1.0 / 19.06.2007
//author:       H.Scheuenstuhl
//modification: Prototyp
//--------------------------------------------------------------------------------
//Beschreibung
//Bits für Maschinentyp und Optionsbit aus iMaPar separieren. Der Maschinen-
//parameter muss wie folgt strukturiert sein:
// Bit   0- 3: Maschinentyp
// Bits  4-15: Optionsbits
AUTHOR : SPAC_slh
FAMILY : GENERAL
NAME : General
VERSION : 1.0
VAR_INPUT
  iMaPar : WORD ;	//auszuwertender Maschinenparameter
END_VAR
VAR_OUTPUT
  oMaTyp : WORD ;	//dekodierter Maschinentyp (1 aus 16)
  oOptBits : WORD ;	//Bit 4-15 von iMaPar (Bit 0-3 nicht belegt)
END_VAR
VAR_TEMP
  svAr1 : DWORD ;
  MaTyp : WORD ;	//dek.Maschinentyp, 1 aus 16
  MaPar : WORD ;
END_VAR
BEGIN
NETWORK
TITLE =
      L     #iMaPar;
      T     #MaPar;
      TAR1  #svAr1;
      LAR1  P##MaTyp;
      L     B#16#0;
      T     #MaTyp;
      L     #MaPar;
      AW    W#16#F;
      JZ    m001;
      +AR1;
      SET;
      S     L [AR1,P#0.0];
m001: LAR1  #svAr1;
      L     #MaTyp;
      T     #oMaTyp;
      L     #MaPar;
      AW    W#16#FFF0;
      T     #oOptBits;
END_FUNCTION

FUNCTION "FC_CK2OP" : VOID	// FC 101
TITLE = Überwachung von 2 Aus-/Eingängen
//________________________________________________________________________________
//$Revision: x.y $
//$Date: 2005/04/26 0:0:0CET $
//$Author: slh $
//$ProjectRevision: Last Checkpoint: m.n $
//
//-------------------------------------------------------------------------------
//*ALL RIGHTS RESERVED
//*Softwareentwicklung
//erstellt: 09.05.2005; Helmut Scheuenstuhl (slh); Scheuenstuhl PAC / V0.1
//Änderung: Datum / Abteilung / Name / Version x.y
//Änderung: 
//        :
//-------------------------------------------------------------------------------
//Beschreibung
//Der Fc dient zur Überwachung von 2 Stellgliedern (Ventile o.ä.)
//Pro Aufruf werden 14 Byte Arbeitsdaten benötigt, deren Adresse über 
//iArbDat(Any) angegeben wird.
//WICHTIGE VORAUSSETZUNG:
//Der Fc arbeitet mit der Plc-Zeit, die mit SFC64 Time_tck ausgelesen und am
//"iAktTime" angeboten werden muß.
AUTHOR : SPAC_slh
FAMILY : Diagnose
NAME : CK2OP
VERSION : 0.1
VAR_INPUT
  iArbDat : ANY ;	//Rettadresse der 14Byte Arbeitsdaten des Fc
  iAktTime : TIME ;	//ausgeleseneSysZeitVonTime_tck SFC64
  iWPaar : TIME ;	//Verzögerung Paarüberwachung, T#0MS= Abwahl
  iWLz : TIME ;	//Verzögerung Laufzeitüberwachung, T#0MS= Abwahl
  iWEndl : TIME ;	//Verzögerung Endlagenüberwachung, T#0MS= Abwahl
  iE1 : BOOL ;	//Schalter, wird durch iA1 angefahren
  iA1 : BOOL ;	//zu überwachender Ausgang 1
  iE2 : BOOL ;	//Schalter, wird durch iA2 angefahren
  iA2 : BOOL ;	//zu überwachender Ausgang 2
  iDL : BOOL ;	//gespeicherte Endstlg.mit Befehl 0 abschalten
  iSq : BOOL ;	//Störung quittieren
  iNoPaar : BOOL ;	//Paarüberwachung abschalten
  iNoLz : BOOL ;	//Laufzeitüberwachung abschalten
  iNoEnd : BOOL ;	//Endlagenüberwachung abschalten
END_VAR
VAR_IN_OUT
  ioFLz1 : BOOL ;	//Laufzeitfehler bei Stlg.1 anfahren
  ioFLz2 : BOOL ;	//Laufzeitfehler bei Stlg.2 anfahren
  ioFEnd1 : BOOL ;	//Fehler:Endlage 1 wurde verlassen
  ioFEnd2 : BOOL ;	//Fehler:Endlage 2 wurde verlassen
  ioFPaar : BOOL ;	//Fehler Paarüberwachung
END_VAR
VAR_TEMP
  AdrArDat : ANY ;	//Übergabeparameter für Adresse der Arbeitsdaten
  svAr1 : DWORD ;
  svAr2 : DWORD ;
  s : UDT 1010;	//stat, da gerettet
  RetVal : INT ;
  Lop1 : BOOL ;
  seEingang : BOOL ;	//SwTimer se Eingang
  seFpEing : BOOL ;	//SwTimer se Eingang pos.Flanke
  seAbgel : BOOL ;	//SwTimer se abgelaufen
  seAusgang : BOOL ;	//SwTimer se Ausgang
  fpiA1 : BOOL ;
  fpiA2 : BOOL ;
  fpSq : BOOL ;	//Flanke Störung quittieren
END_VAR
BEGIN
NETWORK
TITLE = Übergabezeiger für BLKMOV aus iArbDat übernehmen
      TAR1  #svAr1;
      TAR2  #svAr2;
      L     P##iArbDat;
      LAR1;
      LAR2  P##AdrArDat;
      L     W [AR1,P#0.0];
      T     LW [AR2,P#0.0];
      L     D [AR1,P#2.0];
      T     LD [AR2,P#2.0];
      L     D [AR1,P#6.0];
      T     LD [AR2,P#6.0];
      LAR1  #svAr1;
      LAR2  #svAr2;
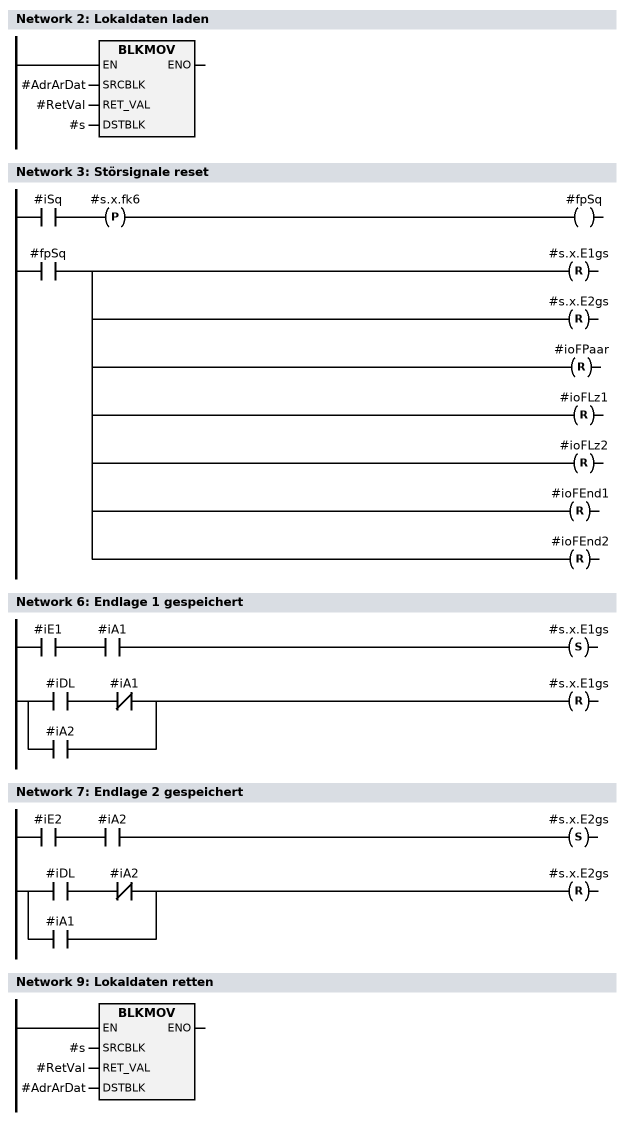
NETWORK
TITLE = Lokaldaten laden
      CALL  "BLKMOV" (
           SRCBLK                   := #AdrArDat,
           RET_VAL                  := #RetVal,
           DSTBLK                   := #s);
      NOP   0;
NETWORK
TITLE = Störsignale reset
      A     #iSq;
      FP    #s.x.fk6;
      =     #fpSq;
      A     #fpSq;
      R     #s.x.E1gs;
      R     #s.x.E2gs;
      R     #ioFPaar;
      R     #ioFLz1;
      R     #ioFLz2;
      R     #ioFEnd1;
      R     #ioFEnd2;
NETWORK
TITLE = Fehler: Paarüberwachung
      L     T#0MS;
      L     #iWPaar;
      ==D;
      O     #iNoPaar;
      JC    t0e1;	//Zeitvorgabe 0ms schaltet Überwachung ab
      R     #seAbgel;
      A     #iE1;
      A     #iE2;
      AN    #fpSq;
      =     #seEingang;
//*** SwZeit ***
      A     #seEingang;
      FP    #s.x.fk0;
      =     #seFpEing;
      AN    #seEingang;
      JC    t0e0;
      L     #iAktTime;
      AN    #seFpEing;
      JC    t0m1;
      T     #s.SwT[0];
t0m1: L     #s.SwT[0];
      -D;
      JPZ   t0m2;
      L     L#2147483647;
      +D;
t0m2: L     #iWPaar;
      >=D;
      =     #seAbgel;
t0e0: A     #seEingang;
      A     #seAbgel;
      =     #seAusgang;
//*** Ende SwZeit ***
      A     #seAusgang;
      S     #ioFPaar;
t0e1: NOP   0;
NETWORK
TITLE = Fehler: Laufzeit
      A     #iA1;
      FP    #s.x.fk4;
      =     #fpiA1;
      A     #iA2;
      FP    #s.x.fk5;
      =     #fpiA2;
      L     T#0MS;
      L     #iWLz;
      ==D;
      O     #iNoLz;
      JC    t1e1;	//Zeitvorgabe 0ms schaltet Überwachung ab
      R     #seAbgel;
      A(;
      AN    #iE1;
      A     #iA1;
      AN    #fpiA1;	//bei direkter Richtungsumschaltung Zeit neu triggern
      AN    #s.x.E1gs;
      O;
      AN    #iE2;
      A     #iA2;
      AN    #fpiA2;	//bei direkter Richtungsumschaltung Zeit neu triggern
      AN    #s.x.E2gs;
      );
      AN    #fpSq;
      =     #seEingang;
//*** SwZeit 1 ***
      A     #seEingang;
      FP    #s.x.fk1;
      =     #seFpEing;
      AN    #seEingang;
      JC    t1e0;
      L     #iAktTime;
      AN    #seFpEing;
      JC    t1m1;
      T     #s.SwT[1];
t1m1: L     #s.SwT[1];
      -D;
      JPZ   t1m2;
      L     L#2147483647;
      +D;
t1m2: L     #iWLz;
      >=D;
      =     #seAbgel;
t1e0: A     #seEingang;
      A     #seAbgel;
      =     #seAusgang;
//*** Ende SwZeit ***
      A     #seAusgang;
      A     #iA1;
      S     #ioFLz1;
      A     #seAusgang;
      A     #iA2;
      S     #ioFLz2;
t1e1: NOP   0;
NETWORK
TITLE = Endlage 1 gespeichert
      A     #iE1;
      A     #iA1;
      S     #s.x.E1gs;
      A(;
      A     #iDL;
      AN    #iA1;
      O     #iA2;
      );
      R     #s.x.E1gs;
      NOP   0;
NETWORK
TITLE = Endlage 2 gespeichert
      A     #iE2;
      A     #iA2;
      S     #s.x.E2gs;
      A(;
      A     #iDL;
      AN    #iA2;
      O     #iA1;
      );
      R     #s.x.E2gs;
      NOP   0;
NETWORK
TITLE = Fehler: Endlage verlassen
      L     T#0MS;
      L     #iWEndl;
      ==D;
      O     #iNoEnd;
      JC    t2e1;	//Zeitvorgabe 0ms schaltet Überwachung ab
      R     #seAbgel;
      A(;
      A     #s.x.E1gs;
      AN    #iE1;
      O;
      A     #s.x.E2gs;
      AN    #iE2;
      );
      AN    #fpSq;
      =     #seEingang;
//*** SwZeit 2 ***
      A     #seEingang;
      FP    #s.x.fk2;
      =     #seFpEing;
      AN    #seEingang;
      JC    t2e0;
      L     #iAktTime;
      AN    #seFpEing;
      JC    t2m1;
      T     #s.SwT[2];
t2m1: L     #s.SwT[2];
      -D;
      JPZ   t2m2;
      L     L#2147483647;
      +D;
t2m2: L     #iWEndl;
      >=D;
      =     #seAbgel;
t2e0: A     #seEingang;
      A     #seAbgel;
      =     #seAusgang;
//*** Ende SwZeit ***
      A     #seAusgang;
      A     #s.x.E1gs;
      AN    #iE1;
      S     #ioFEnd1;
      A     #seAusgang;
      A     #s.x.E2gs;
      AN    #iE2;
      S     #ioFEnd2;
t2e1: NOP   0;
NETWORK
TITLE = Lokaldaten retten
      CALL  "BLKMOV" (
           SRCBLK                   := #s,
           RET_VAL                  := #RetVal,
           DSTBLK                   := #AdrArDat);
      NOP   0;
END_FUNCTION

FUNCTION "FC_CK1OP" : VOID	// FC 102
TITLE = Überwachung von 1 Aus-/Eingang
//________________________________________________________________________________
//$Revision: x.y $
//$Date: 2005/04/26 0:0:0CET $
//$Author: slh $
//$ProjectRevision: Last Checkpoint: m.n $
//
//-------------------------------------------------------------------------------
//*ALL RIGHTS RESERVED
//*Softwareentwicklung
//erstellt: 09.05.2005; Helmut Scheuenstuhl (slh); Scheuenstuhl PAC / V0.1
//Änderung: Datum / Abteilung / Name / Version x.y
//Änderung: 
//        :
//-------------------------------------------------------------------------------
//Beschreibung
//Der Fc dient zur Überwachung von 1 Stellglied (Ventile o.ä.)
//Pro Aufruf werden 14 Byte Arbeitsdaten benötigt, deren Adresse über 
//iArbDat(Any) angegeben wird.
//WICHTIGE VORAUSSETZUNG:
//Der Fc arbeitet mit der Plc-Zeit, die mit SFC64 Time_tck ausgelesen und am
//"iAktTime" angeboten werden muß.
AUTHOR : SPAC_slh
FAMILY : Diagnose
NAME : CK1OP
VERSION : 0.1
VAR_INPUT
  iArbDat : ANY ;	//Rettadresse der 14Byte Arbeitsdaten des Fc
  iAktTime : TIME ;	//ausgeleseneSysZeitVonTime_tck SFC64
  iWAus : TIME ;	//Verzögerung Ausschaltüberwachung, T#0MS= Abwahl
  iWEin : TIME ;	//Verzögerung Einschaltüberwachung, T#0MS= Abwahl
  iWUnt : TIME ;	//Verzögerung Unterbrechungsüberwachung, T#0MS= Abwahl
  iE1 : BOOL ;	//Schalter, wird durch iA1 angefahren
  iA1 : BOOL ;	//zu überwachender Ausgang 1
  iSq : BOOL ;	//Störung quittieren
END_VAR
VAR_IN_OUT
  ioFEin : BOOL ;	//Fehler Einschaltüberwachung
  ioFUnt : BOOL ;	//Fehler:Unterbrechungsüberwachung
  ioFAus : BOOL ;	//Fehler Ausschaltüberwachung
END_VAR
VAR_TEMP
  AdrArDat : ANY ;	//Übergabeparameter für Adresse der Arbeitsdaten
  svAr1 : DWORD ;
  svAr2 : DWORD ;
  s : UDT 1010;	//stat, da gerettet
  RetVal : INT ;
  Lop1 : BOOL ;
  seEingang : BOOL ;	//SwTimer se Eingang
  seFpEing : BOOL ;	//SwTimer se Eingang pos.Flanke
  seAbgel : BOOL ;	//SwTimer se abgelaufen
  seAusgang : BOOL ;	//SwTimer se Ausgang
  fpiA1 : BOOL ;
  fpSq : BOOL ;	//Flanke Störung quittieren
END_VAR
BEGIN
NETWORK
TITLE = Übergabezeiger für BLKMOV aus iArbDat übernehmen
      TAR1  #svAr1;
      TAR2  #svAr2;
      L     P##iArbDat;
      LAR1;
      LAR2  P##AdrArDat;
      L     W [AR1,P#0.0];
      T     LW [AR2,P#0.0];
      L     D [AR1,P#2.0];
      T     LD [AR2,P#2.0];
      L     D [AR1,P#6.0];
      T     LD [AR2,P#6.0];
      LAR1  #svAr1;
      LAR2  #svAr2;
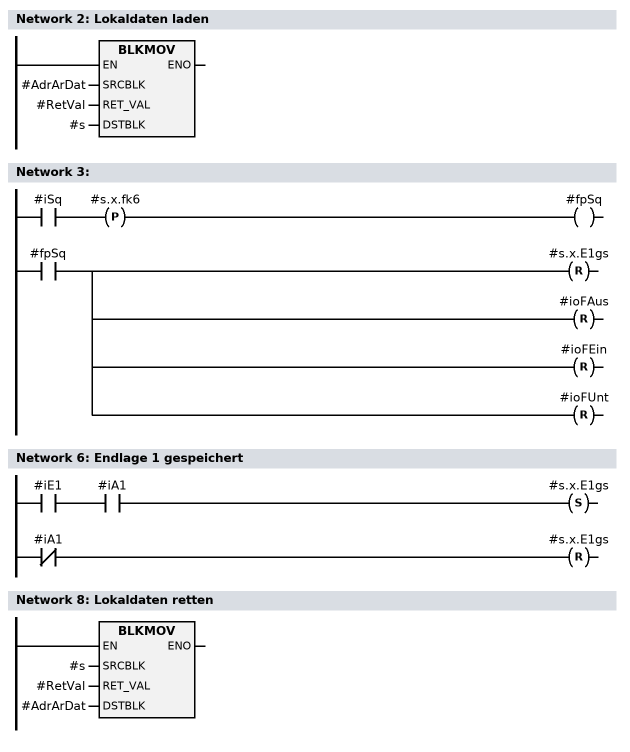
NETWORK
TITLE = Lokaldaten laden
      CALL  "BLKMOV" (
           SRCBLK                   := #AdrArDat,
           RET_VAL                  := #RetVal,
           DSTBLK                   := #s);
      NOP   0;
NETWORK
TITLE =
      A     #iSq;
      FP    #s.x.fk6;
      =     #fpSq;
      A     #fpSq;
      R     #s.x.E1gs;
      R     #ioFAus;
      R     #ioFEin;
      R     #ioFUnt;
NETWORK
TITLE = Fehler: Ausschaltüberwachung
      L     T#0MS;
      L     #iWAus;
      ==D;
      JC    t0e1;	//Zeitvorgabe 0ms schaltet Überwachung ab
      R     #seAbgel;
      A     #iE1;
      AN    #iA1;
      AN    #fpSq;
      =     #seEingang;
//*** SwZeit ***
      A     #seEingang;
      FP    #s.x.fk0;
      =     #seFpEing;
      AN    #seEingang;
      JC    t0e0;
      L     #iAktTime;
      AN    #seFpEing;
      JC    t0m1;
      T     #s.SwT[0];
t0m1: L     #s.SwT[0];
      -D;
      JPZ   t0m2;
      L     L#2147483647;
      +D;
t0m2: L     #iWAus;
      >=D;
      =     #seAbgel;
t0e0: A     #seEingang;
      A     #seAbgel;
      =     #seAusgang;
//*** Ende SwZeit ***
      A     #seAusgang;
      S     #ioFAus;
t0e1: NOP   0;
NETWORK
TITLE = Fehler: Laufzeit, Einschaltüberwachung
      A     #iA1;
      FP    #s.x.fk4;
      =     #fpiA1;
      L     T#0MS;
      L     #iWEin;
      ==D;
      JC    t1e1;	//Zeitvorgabe 0ms schaltet Überwachung ab
      R     #seAbgel;
      AN    #iE1;
      A     #iA1;
      AN    #s.x.E1gs;
      AN    #fpSq;
      =     #seEingang;
//*** SwZeit 1 ***
      A     #seEingang;
      FP    #s.x.fk1;
      =     #seFpEing;
      AN    #seEingang;
      JC    t1e0;
      L     #iAktTime;
      AN    #seFpEing;
      JC    t1m1;
      T     #s.SwT[1];
t1m1: L     #s.SwT[1];
      -D;
      JPZ   t1m2;
      L     L#2147483647;
      +D;
t1m2: L     #iWEin;
      >=D;
      =     #seAbgel;
t1e0: A     #seEingang;
      A     #seAbgel;
      =     #seAusgang;
//*** Ende SwZeit ***
      A     #seAusgang;
      S     #ioFEin;
t1e1: NOP   0;
NETWORK
TITLE = Endlage 1 gespeichert
      A     #iE1;
      A     #iA1;
      S     #s.x.E1gs;
      AN    #iA1;
      R     #s.x.E1gs;
      NOP   0;
NETWORK
TITLE = Fehler: Endlage verlassen=Unterbrechungsüberwachung
      L     T#0MS;
      L     #iWUnt;
      ==D;
      JC    t2e1;	//Zeitvorgabe 0ms schaltet Überwachung ab
      R     #seAbgel;
      A     #s.x.E1gs;
      AN    #iE1;
      AN    #fpSq;
      =     #seEingang;
//*** SwZeit 2 ***
      A     #seEingang;
      FP    #s.x.fk2;
      =     #seFpEing;
      AN    #seEingang;
      JC    t2e0;
      L     #iAktTime;
      AN    #seFpEing;
      JC    t2m1;
      T     #s.SwT[2];
t2m1: L     #s.SwT[2];
      -D;
      JPZ   t2m2;
      L     L#2147483647;
      +D;
t2m2: L     #iWUnt;
      >=D;
      =     #seAbgel;
t2e0: A     #seEingang;
      A     #seAbgel;
      =     #seAusgang;
//*** Ende SwZeit ***
      A     #seAusgang;
      A     #s.x.E1gs;
      AN    #iE1;
      S     #ioFUnt;
t2e1: NOP   0;
NETWORK
TITLE = Lokaldaten retten
      CALL  "BLKMOV" (
           SRCBLK                   := #s,
           RET_VAL                  := #RetVal,
           DSTBLK                   := #AdrArDat);
      NOP   0;
END_FUNCTION

FUNCTION "INPUT_MASTER" : VOID	// FC 111
TITLE = EINGÄNGE VOM MASTERSYSTEM LESEN
//Die Kommunikation mit dem Mastersystem erfolgt durch Merkerwörter
AUTHOR : APetz
VERSION : 0.1
VAR_TEMP
  B_TEMP : BYTE ;	//Zwischenspeicher
  X_TEMP : BOOL ;	//Zwischenspeicher
END_VAR
BEGIN
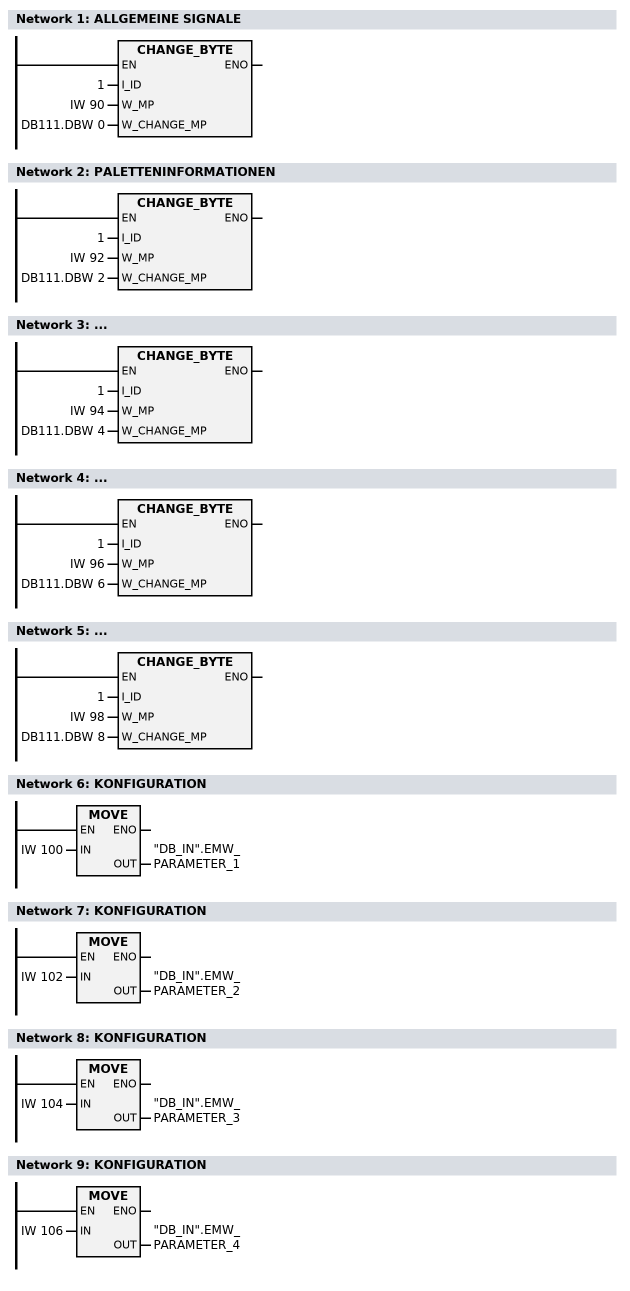
NETWORK
TITLE = ALLGEMEINE SIGNALE
//Eingangswort in Datenbaustein transferieren
//EW90 (aus HW-Konfiguration) nach DB111.DBW0 schreiben (Byte-/Bitzugriff)
//HINWEIS: Das Tauschen der Bytes wird, durch die unterschiedlichen Notationen,
//         benötigt.
      CALL  "CHANGE_BYTE" (
           I_ID                     := 1,
           W_MP                     := IW 90,
           W_CHANGE_MP              := DB111.DBW 0);	// aus Konfiguration
      NOP   0;
NETWORK
TITLE = PALETTENINFORMATIONEN
//Eingangswort in Datenbaustein transferieren
//EW92 (aus HW-Konfiguration) nach DB111.DBW2 schreiben (Byte-/Bitzugriff)
//HINWEIS: Das Tauschen der Bytes wird, durch die unterschiedlichen Notationen,
//         benötigt.
      CALL  "CHANGE_BYTE" (
           I_ID                     := 1,
           W_MP                     := IW 92,
           W_CHANGE_MP              := DB111.DBW 2);
      NOP   0;
NETWORK
TITLE = ...
//Eingangswort in Datenbaustein transferieren
//EW94 (aus HW-Konfiguration) nach DB111.DBW4 schreiben (Byte-/Bitzugriff)
//HINWEIS: Das Tauschen der Bytes wird, durch die unterschiedlichen Notationen,
//         benötigt.
      CALL  "CHANGE_BYTE" (
           I_ID                     := 1,
           W_MP                     := IW 94,
           W_CHANGE_MP              := DB111.DBW 4);
      NOP   0;
NETWORK
TITLE = ...
//Eingangswort in Datenbaustein transferieren
//EW96 (aus HW-Konfiguration) nach DB111.DBW6 schreiben (Byte-/Bitzugriff)
//HINWEIS: Das Tauschen der Bytes wird, durch die unterschiedlichen Notationen,
//         benötigt.
      CALL  "CHANGE_BYTE" (
           I_ID                     := 1,
           W_MP                     := IW 96,
           W_CHANGE_MP              := DB111.DBW 6);
      NOP   0;
NETWORK
TITLE = ...
//Eingangswort in Datenbaustein transferieren
//EW98 (aus HW-Konfiguration) nach DB111.DBW8 schreiben (Byte-/Bitzugriff)
//HINWEIS: Das Tauschen der Bytes wird, durch die unterschiedlichen Notationen,
//         benötigt.
      CALL  "CHANGE_BYTE" (
           I_ID                     := 1,
           W_MP                     := IW 98,
           W_CHANGE_MP              := DB111.DBW 8);
      NOP   0;
NETWORK
TITLE = KONFIGURATION
//Eingangswort in Datenbaustein transferieren
//EW100 (aus HW-Konfiguration) nach DB111.DBW10 schreiben (Wort)
      L     IW 100;
      T     "DB_IN".EMW_PARAMETER_1;
      NOP   0;
NETWORK
TITLE = KONFIGURATION
//Eingangswort in Datenbaustein transferieren
//EW102 (aus HW-Konfiguration) nach DB111.DBW12 schreiben (Wort)
      L     IW 102;
      T     "DB_IN".EMW_PARAMETER_2;
      NOP   0;
NETWORK
TITLE = KONFIGURATION
//Eingangswort in Datenbaustein transferieren
//EW104 (aus HW-Konfiguration) nach DB111.DBW14 schreiben (Wort)
      L     IW 104;
      T     "DB_IN".EMW_PARAMETER_3;
      NOP   0;
NETWORK
TITLE = KONFIGURATION
//Eingangswort in Datenbaustein transferieren
//EW106 (aus HW-Konfiguration) nach DB111.DBW16 schreiben (Wort)
      L     IW 106;
      T     "DB_IN".EMW_PARAMETER_4;
      NOP   0;
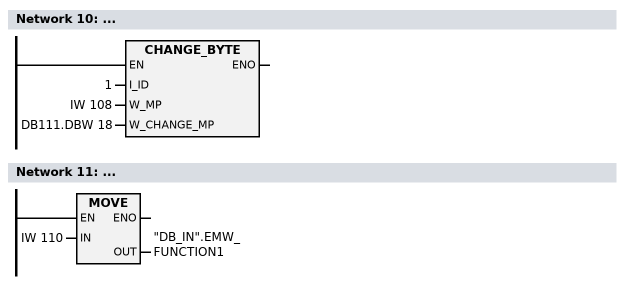
NETWORK
TITLE = ...
//Eingangswort in Datenbaustein transferieren
//EW108 (aus HW-Konfiguration) nach DB111.DBW18 schreiben (Byte-/Bitzugriff)
//HINWEIS: Das Tauschen der Bytes wird, durch die unterschiedlichen Notationen,
//         benötigt.
      CALL  "CHANGE_BYTE" (
           I_ID                     := 1,
           W_MP                     := IW 108,
           W_CHANGE_MP              := DB111.DBW 18);
      NOP   0;
NETWORK
TITLE = ...
//Eingangswort in Datenbaustein transferieren
//EW110 (aus HW-Konfiguration) nach DB111.DBW20 schreiben (Wort)
//
      L     IW 110;
      T     "DB_IN".EMW_FUNCTION1;
      NOP   0;
END_FUNCTION

FUNCTION "OUTPUT_MASTER" : VOID	// FC 112
TITLE = AUSGÄNGE AN MASTERSYSTEM SCHREIBEN
//Die Kommunikation mit dem Mastersystem erfolgt durch Merkerwörter
AUTHOR : APetz
VERSION : 0.1
BEGIN
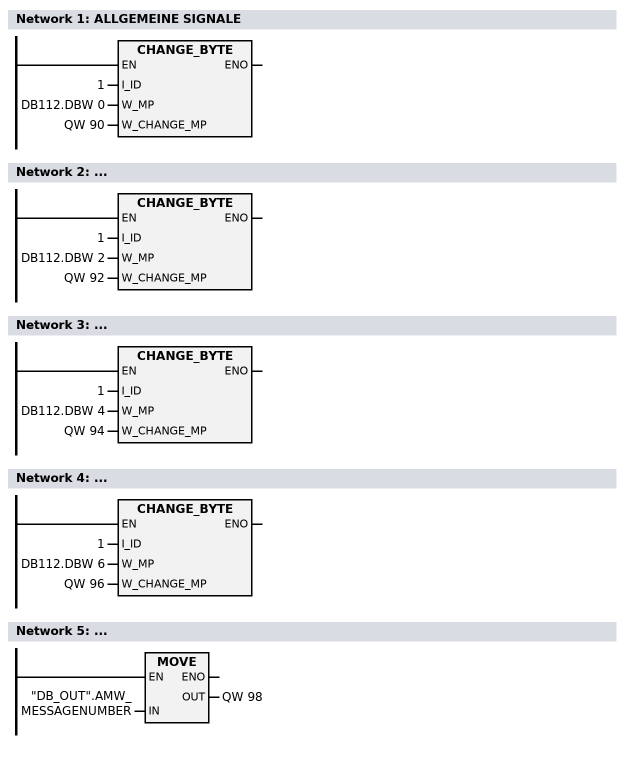
NETWORK
TITLE = ALLGEMEINE SIGNALE
//Datenbaustein nach Ausgangswort transferieren
//DB112.DBW0 nach AW90 (HW-Konfiguration) schreiben (Byte-/Bitzugriff)
//HINWEIS: Das Tauschen der Bytes wird, durch die unterschiedlichen Notationen,
//         benötigt.
      CALL  "CHANGE_BYTE" (
           I_ID                     := 1,
           W_MP                     := DB112.DBW 0,
           W_CHANGE_MP              := QW 90);
      NOP   0;
NETWORK
TITLE = ...
//Datenbaustein nach Ausgangswort transferieren
//DB112.DBW2 nach AW92 (HW-Konfiguration) schreiben (Byte-/Bitzugriff)
//HINWEIS: Das Tauschen der Bytes wird, durch die unterschiedlichen Notationen,
//         benötigt.
      CALL  "CHANGE_BYTE" (
           I_ID                     := 1,
           W_MP                     := DB112.DBW 2,
           W_CHANGE_MP              := QW 92);
      NOP   0;
NETWORK
TITLE = ...
//Datenbaustein nach Ausgangswort transferieren
//DB112.DBW4 nach AW94 (HW-Konfiguration) schreiben (Byte-/Bitzugriff)
//HINWEIS: Das Tauschen der Bytes wird, durch die unterschiedlichen Notationen,
//         benötigt.
      CALL  "CHANGE_BYTE" (
           I_ID                     := 1,
           W_MP                     := DB112.DBW 4,
           W_CHANGE_MP              := QW 94);
      NOP   0;
NETWORK
TITLE = ...
//Datenbaustein nach Ausgangswort transferieren
//DB112.DBW6 nach AW96 (HW-Konfiguration) schreiben (Byte-/Bitzugriff)
//HINWEIS: Das Tauschen der Bytes wird, durch die unterschiedlichen Notationen,
//         benötigt.
      CALL  "CHANGE_BYTE" (
           I_ID                     := 1,
           W_MP                     := DB112.DBW 6,
           W_CHANGE_MP              := QW 96);
      NOP   0;
NETWORK
TITLE = ...
//Datenbaustein nach Ausgangswort transferieren
//DB112.DBW8 nach AW98 (HW-Konfiguration) schreiben (Byte-/Bitzugriff)
//HINWEIS: Das Tauschen der Bytes wird, durch die unterschiedlichen Notationen,
//         benötigt.
      L     "DB_OUT".AMW_MESSAGENUMBER;
      T     QW 98;
      NOP   0;
END_FUNCTION

FUNCTION "CallAutoSusDoor" : VOID	// FC 120
TITLE = AUFRUF AUTOMATISCHE RÜSTPLATZTÜREN
//------------------------------------------------------------------------------
//version:      1.0 / 24.09.2007
//author:       A.Petz
//modification: Prototyp
//-------------------------------------------------------------------------------
//Einstellungen und Auswertungen für automatische (pneum.) Rüstplatztüren
AUTHOR : APetz
FAMILY : AUTOMAT
NAME : SusDoor
VERSION : 1.0
VAR_TEMP
  LocInt1 : INT ;	//lokalVariable0
  LocInt2 : INT ;	//lokalVariable1
  LocInt3 : INT ;	//lokalVariable2
  ParameterMsb : BYTE ;	//Parametereintrag (1000er und 100er)
  ParameterLsb : BYTE ;	//Parametereintrag (10er und 1er)
  Parameter10e0 : BYTE ;	//Parametereintrag (Einer)
  Parameter10e1 : BYTE ;	//Parametereintrag (Zehner)
  Parameter10e2 : BYTE ;	//Parametereintrag (Hunderter)
  Parameter10e3 : BYTE ;	//Parametereintrag (Tausender)
  ModuleEnable : BOOL ;	//Bausteinfreigabe (Sammelstörung)
  CompareMaParValue : BOOL ;	//Vergleich Maschinenparameter: Wert in Dekade positiv
  LocM0 : BOOL ;	//lokaler Operationsmerker0
END_VAR
BEGIN
NETWORK
TITLE = ENABLE-Eingang prüfen
//Auswerten des BIE-Statusbit. Dieses entspricht dem EN (ENABLE)-Einganges bei 
//KOP/FUP. Wenn EN=FALSE dann verlasse Baustein.
//
      AN    BR;
      SAVE;
      BEC;
NETWORK
TITLE = Bausteinfreigabe
//Fehlerauswertung Baustein intern:
//Bausteinfreigabe wird gesetzt
      A     "M_HIGH";
      =     L 10.0;
NETWORK
TITLE = Funktionsweise ZPS aus Maschinenparameter lesen
//Daten aus Maschinenparameter extrahieren
      CALL  "FUNCTIONS" (
           iMaPar                   := "DB_IN".EMW_PARAMETER_3,
           iDekade                  := B#16#0,
           iVglWert                 := B#16#0,
           oMsb                     := #LocInt3,
           oLsb                     := LB 5,
           o10e0                    := #ParameterMsb,
           o10e1                    := #ParameterLsb,
           o10e2                    := #Parameter10e0,
           o10e3                    := #Parameter10e1,
           oVglTrue                 := L 10.1);
      NOP   0;
NETWORK
TITLE = Typumwandlung der Bausteinparameter
      A     "M_HIGH";
      =     L 11.0;
      A     L 11.0;
      JNB   _001;
      L     #ParameterLsb;
      T     #LocInt1;
_001: NOP   0;
      A     L 11.0;
      JNB   _002;
      L     #Parameter10e0;
      T     #LocInt2;
_002: NOP   0;
NETWORK
TITLE =
      A(;
      L     #LocInt1;
      L     1;
      ==I;
      );
      =     L 11.0;
      BLD   103;
      A(;
      L     #LocInt2;
      L     1;
      ==I;
      );
      =     L 11.1;
      BLD   103;
      A     "M_HIGH";
      A     "mTypeDMCxxU2";
      JNB   M002;
      CALL  "AutoSusDoor" , DB 20 (
           iMode                    := #ParameterMsb,
           iSafetyEdgeMonitoringTim := B#16#15,
           iOnly1SusDoor            := L 11.0,
           iAutoReverse             := L 11.1);
M002: NOP   0;
NETWORK
TITLE = Bausteinfreigabe
//Statusbit BIE=ENO setzen, wenn Funktion ohne Fehler durchlaufen wurde.
      A     L 10.0;
      SAVE;
END_FUNCTION

FUNCTION "INPUT_PERIPHERIE" : VOID	// FC 121
TITLE = EINGÄNGE VOM PERPHERIE LESEN
//Eingangssignale von Peripherie (ET200S) rangieren
AUTHOR : APetz
VERSION : 0.1
VAR_TEMP
  ModuleEnable : BOOL ;	//Bausteinfreigabe - Sammelstörung
END_VAR
BEGIN
NETWORK
TITLE = ENABLE-Eingang prüfen
//Auswerten des BIE-Statusbit. Dieses entspricht dem EN (ENABLE)-Einganges bei 
//KOP/FUP. Wenn EN=FALSE dann verlasse Baustein.
//
      AN    BR;
      SAVE;
      BEC;
NETWORK
TITLE = BAUSTEINFREIGABE
//Fehlerauswertung Baustein intern:
//Bausteinfreigabe wird gesetzt
      A     "M_HIGH";
      =     #ModuleEnable;
NETWORK
TITLE = Rangierer
      A     I 2.0;
      =     "EpxSusDoorSystPressMax";
      A     I 2.1;
      =     "EpxCloseSusDoor";
      A     I 2.2;
      =     "EpxOpenSusDoor";
      A     I 2.3;
      =     "EpxRobotLock";
      A     I 3.0;
      =     "EpxSafetyEdgeSusDoor";
      A     I 3.1;
      =     "EpxSusDoorPressMonOpen";
      A     I 3.2;
      =     "EpxSusDoorPressMonClose";
      A     I 4.0;
      =     "EpxSusDoorLeftOpen";
      A     I 4.1;
      =     "EpxSusDoorRightOpen";
      A     I 4.2;
      =     "EpxSusDoorClosed";
      A     I 4.3;
      =     "EpxSusDoorClosedLocked";
NETWORK
TITLE = BAUSTEINFREIGABE
//Statusbit BIE=ENO setzen, wenn Funktion ohne Fehler durchlaufen wurde.
      A     #ModuleEnable;
      SAVE;
END_FUNCTION

FUNCTION "OUTPUT_PERIPHERIE" : VOID	// FC 122
TITLE = AUSGÄNGE AN PERIPHERIE SCHREIBEN
//Ausgangssignale an Peripherie (ET200S) rangieren
AUTHOR : APetz
VERSION : 0.1
VAR_TEMP
  ModuleEnable : BOOL ;	//Bausteinfreigabe - Sammelstörung
END_VAR
BEGIN
NETWORK
TITLE = ENABLE-Eingang prüfen
//Auswerten des BIE-Statusbit. Dieses entspricht dem EN (ENABLE)-Einganges bei 
//KOP/FUP. Wenn EN=FALSE dann verlasse Baustein.
//
      AN    BR;
      SAVE;
      BEC;
NETWORK
TITLE = BAUSTEINFREIGABE
//Fehlerauswertung Baustein intern:
//Bausteinfreigabe wird gesetzt
      A     "M_HIGH";
      =     #ModuleEnable;
NETWORK
TITLE = Rangierer
      A     "ApxMainValveSusDoor";
      =     Q 6.0;
      A     "ApxCloseSusDoor";
      =     Q 6.1;
      A     "ApxOpenSusDoor";
      =     Q 6.2;
NETWORK
TITLE = BAUSTEINFREIGABE
//Statusbit BIE=ENO setzen, wenn Funktion ohne Fehler durchlaufen wurde.
      A     #ModuleEnable;
      SAVE;
END_FUNCTION

DATA_BLOCK "DB_Message"	// DB 2
AUTHOR : SPAC_slh
VERSION : 0.1
  STRUCT
   ALARM_001 : BOOL ;	//Schaltschranktemperatur zu hoch
   ALARM_002 : BOOL ;	//Schaltschranktemperatur - Grenzwert überschritten
   F003 : BOOL ;	//1-
   F004 : BOOL ;	//1-
   F005 : BOOL ;	//1-
   F006 : BOOL ;	//1-
   F007 : BOOL ;	//1-
   F008 : BOOL ;	//1-
   F009 : BOOL ;	//1-
   F010 : BOOL ;	//1-
   F011 : BOOL ;	//1-
   F012 : BOOL ;	//1-
   F013 : BOOL ;	//1-
   F014 : BOOL ;	//1-
   F015 : BOOL ;	//1-
   F016 : BOOL ;	//1-
   ALARM_017 : BOOL ;	//Nullpunktspannsysten Zeitüberschreitung beim Lösen[1]
   ALARM_018 : BOOL ;	//Nullpunktspannsysten Zeitüberschreitung beim Spannen[1]
   ALARM_019 : BOOL ;	//Nullpunktspannsystem Druck am Druckschalter[1]-Maximum nicht vorhanden
   ALARM_020 : BOOL ;	//Nullpunktspannsystem Druck am Druckschalter[1]-Minimum zu hoch
   ALARM_021 : BOOL ;	//Nullpunktspannsystem Signale an Druckschaltern[1] nicht korrekt (Plausibilität)
   ALARM_022 : BOOL ;	//Nullpunktspannsysten Zeitüberschreitung beim Lösen[2]
   ALARM_023 : BOOL ;	//Nullpunktspannsysten Zeitüberschreitung beim Spannen[2]
   ALARM_024 : BOOL ;	//Nullpunktspannsystem Druck am Druckschalter[2]-Maximum nicht vorhanden
   ALARM_025 : BOOL ;	//Nullpunktspannsystem Druck am Druckschalter[2]-Minimum zu hoch
   ALARM_026 : BOOL ;	//Nullpunktspannsystem Signale an Druckschaltern[2] nicht korrekt (Plausibilität)
   ALARM_027 : BOOL ;	//Nullpunktspannsysten Zeitüberschreitung beim Aktivieren der Auflagenkontrolle
   ALARM_028 : BOOL ;	//Nullpunktspannsysten Zeitüberschreitung beim Abschalten der Auflagenkontrolle
   ALARM_029 : BOOL ;	//Nullpunktspannsystem Staudruck für Auflagenkontrolle nicht vorhanden
   ALARM_030 : BOOL ;	//Nullpunktspannsystem Staudruck für Auflagenkontrolle nicht Minimum
   ALARM_031 : BOOL ;	//Nullpunktspannsystem Signale am Auflagenkontrolle nicht korrekt (Plausibilität)
   ALARM_032 : BOOL ;	//Nullpunktspannsysten Zeitüberschreitung beim Aktivieren der Verriegelungskontr.
   ALARM_033 : BOOL ;	//Nullpunktspannsysten Zeitüberschreitung beim Abschalten der Verriegelungskontr.
   ALARM_034 : BOOL ;	//Nullpunktspannsystem Druck an Verriegelungskontrolle nicht vorhanden
   ALARM_035 : BOOL ;	//Nullpunktspannsystem Druck an Verriegelungskontrolle nicht Minimum
   ALARM_036 : BOOL ;	//Nullpunktspannsystem Signale an Verriegelunkontr. nicht korrekt (Plausibilität)
   ALARM_037 : BOOL ;	//Nullpunktspannsystem nicht korrekt gespannt /Freigabe PW nicht möglich
   ALARM_038 : BOOL ;	//Nullpunktspannsystem nicht korrekt gespannt /Verfahren der Achsen nicht möglich
   ALARM_039 : BOOL ;	//Nullpunktspannsystem Lösen nicht möglich
   F040 : BOOL ;	//1-
   F041 : BOOL ;	//1-
   F042 : BOOL ;	//1-
   F043 : BOOL ;	//1-
   F044 : BOOL ;	//1-
   F045 : BOOL ;	//1-
   F046 : BOOL ;	//1-
   F047 : BOOL ;	//1-
   F048 : BOOL ;	//1-
   ALARM_049 : BOOL ;	//Hydraulikfilter Maschine verschmutzt
   ALARM_050 : BOOL ;	//HYD: Hydrauliktemperatur Maschine überschritten
   F051 : BOOL ;	//1-
   F052 : BOOL ;	//1-
   F053 : BOOL ;	//1-
   F054 : BOOL ;	//1-
   F055 : BOOL ;	//1-
   F056 : BOOL ;	//1-
   F057 : BOOL ;	//1-
   F058 : BOOL ;	//1-
   F059 : BOOL ;	//1-
   F060 : BOOL ;	//1-
   F061 : BOOL ;	//1-
   F062 : BOOL ;	//1-
   F063 : BOOL ;	//1-
   F064 : BOOL ;	//1-
   ALARM_065 : BOOL ;	//Störung in Energieversorgung Nebel-u.Rauchabscheider_1
   ALARM_066 : BOOL ;	//Störung in Energieversorgung Nebel-u.Rauchabscheider_2
   F067 : BOOL ;	//1-
   F068 : BOOL ;	//1-
   F069 : BOOL ;	//1-
   F070 : BOOL ;	//1-
   F071 : BOOL ;	//1-
   F072 : BOOL ;	//1-
   F073 : BOOL ;	//1-
   F074 : BOOL ;	//1-
   F075 : BOOL ;	//1-
   F076 : BOOL ;	//1-
   F077 : BOOL ;	//1-
   F078 : BOOL ;	//1-
   F079 : BOOL ;	//1-
   F080 : BOOL ;	//1-
   ALARM_081 : BOOL ;	//Vakuumspannsystem Zeitüberschreitung beim Lösen (Arbeitsraum)
   ALARM_082 : BOOL ;	//Vakuumspannsystem Zeitüberschreitung beim Spannen (Arbeitsraum)
   ALARM_083 : BOOL ;	//Vakuumspannsystem Druck am Druckschalter-Maximum nicht vorhanden (Arbeitsraum)
   ALARM_084 : BOOL ;	//Vakuumspannsystem Druck am Druckschalter-Minimum zu hoch (Arbeitsraum)
   ALARM_085 : BOOL ;	//Vakuumspannsystem Signale an Druckschaltern nicht korrekt-Plausibilität (ARB)
   ALARM_086 : BOOL ;	//Vakuumspannsystem im Arbeitsraum nicht Betriebsbereit (z.B.Störung der Energie)
   ALARM_087 : BOOL ;	//Vakuumspannsystem am Rüstplatz nicht Betriebsbereit (z.B.Störung der Energie)
   ALARM_088 : BOOL ;	//Vakuumspannsystem Zeitüberschreitung beim Lösen (Rüstplatz)
   ALARM_089 : BOOL ;	//Vakuumspannsystem Zeitüberschreitung beim Spannen (Rüstplatz)
   ALARM_090 : BOOL ;	//Vakuumspannsystem Druck am Druckschalter-Minimum zu hoch (Rüstplatz)
   ALARM_091 : BOOL ;	//Vakuumspannsystem Druck am Druckschalter-Maximum nicht vorhanden (Rüstplatz)
   ALARM_092 : BOOL ;	//Vakuumspannsystem Signale an Druckschaltern nicht korrekt-Plausibilität (RPL)
   F093 : BOOL ;	//1-
   F094 : BOOL ;	//1-
   F095 : BOOL ;	//1-
   F096 : BOOL ;	//1-
   ALARM_097 : BOOL ;	//Km-Hautpventil nicht offen, E9.0 meldet "zu", muss 0-Signal melden
   ALARM_098 : BOOL ;	//Km-Hautpventil schließt nicht, E9.0 muss 1-Signal melden
   ALARM_099 : BOOL ;	//WHG-Alarm
   ALARM_100 : BOOL ;	//minimaler Füllstand in KSA erreicht
   ALARM_101 : BOOL ;	//Km-Systemdruck fehlt, E8.3 muss 1-Signal melden
   ALARM_102 : BOOL ;	//Km-Systemdruck, Druckschalter defekt, E8.3 muss 0-Signal melden
   ALARM_103 : BOOL ;	//Km-Durchfluss fehlt, E9.2 muss 1-Signal melden
   ALARM_104 : BOOL ;	//Km-Durchfluss-Schalter defekt, E9.2 muss 0-Signal melden
   ALARM_105 : BOOL ;	//Kühlmittelfeinfilter verschmutzt E10.1
   ALARM_106 : BOOL ;	//Kühlmittelfeinfilter Schalterpaarüberwachung E10.1/E102
   F107 : BOOL ;	//1-
   F108 : BOOL ;	//1-
   F109 : BOOL ;	//1-
   F110 : BOOL ;	//1-
   F111 : BOOL ;	//1-
   F112 : BOOL ;	//1-
   ALARM_113 : BOOL ;	//Zeitüberschreitung beim Aktivieren der KSS-Zufuhr (Niederdruck)
   ALARM_114 : BOOL ;	//Funktionsüberwachung Strömungssensor - Unterbrechung (Niederdruck)
   ALARM_115 : BOOL ;	//Zeitüberschreitung beim Abschalten der KSS-Zufuhr (Niederdruck)
   ALARM_116 : BOOL ;	//Leitungsüberwachung Strömungssensor (Niederdruck)
   ALARM_117 : BOOL ;	//Zeitüberschreitung beim Aktivieren der KSS-Zufuhr (Hochdruck)
   ALARM_118 : BOOL ;	//Funktionsüberwachung Strömungssensor - Unterbrechung (Hochdruck)
   ALARM_119 : BOOL ;	//Zeitüberschreitung beim Abschalten der KSS-Zufuhr (Hochdruck)
   ALARM_120 : BOOL ;	//Leitungsüberwachung Strömungssensor (Hochdruck)
   F121 : BOOL ;	//1-
   F122 : BOOL ;	//1-
   F123 : BOOL ;	//1-
   F124 : BOOL ;	//1-
   F125 : BOOL ;	//1-
   F126 : BOOL ;	//1-
   F127 : BOOL ;	//1-
   F128 : BOOL ;	//1-
   ALARM_129 : BOOL ;	//Spannsystem Zeitüberschreitung beim SysDruck für Lösen aktivieren[1]
   ALARM_130 : BOOL ;	//Spannsystem Zeitüberschreitung beim Spannen[1]
   ALARM_131 : BOOL ;	//Spannsystem Systemdruck für Lösen [1]-Maximum nicht vorhanden
   ALARM_132 : BOOL ;	//Spannsystem Systemdruck für Lösen [1]-Minimum,Restdruck vorhanden
   ALARM_133 : BOOL ;	//Spannsystem Signale an Druckschaltern[1] nicht korrekt (Plausibilität)
   ALARM_134 : BOOL ;	//Spannsystem Zeitüberschreitung beim Lösen[2]
   ALARM_135 : BOOL ;	//Spannsystem Zeitüberschreitung beim Spannen[2]
   ALARM_136 : BOOL ;	//Spannsystem nicht gelöst[2], Endlage verlassen
   ALARM_137 : BOOL ;	//Spannsystem nicht gespannt[2], Endlage verlassen
   ALARM_138 : BOOL ;	//Spannsystem Signale an Druckschaltern[2] nicht korrekt (Plausibilität)
   ALARM_139 : BOOL ;	//Spannsystem Zeitüberschreitung beim Aktivieren der Auflagenkontrolle
   ALARM_140 : BOOL ;	//Spannsystem Zeitüberschreitung beim Abschalten der Auflagenkontrolle
   ALARM_141 : BOOL ;	//Spannsystem Staudruck für Auflagenkontrolle nicht vorhanden
   ALARM_142 : BOOL ;	//Spannsystem Staudruck für Auflagenkontrolle nicht Minimum
   ALARM_143 : BOOL ;	//Spannsystem Signale am Auflagenkontrolle nicht korrekt (Plausibilität)
   ALARM_144 : BOOL ;	//Spannsystem spannen mit Wkst.aber Schalter "gespannt ohne Wkst"=log.1
   ALARM_145 : BOOL ;	//Spannsystem Schalterpaarüberwachung gelöst:Druck vorhanden/drucklos
   ALARM_146 : BOOL ;	//Spannsystem Schalterpaarüberwachung gespannt:Druck vorhanden/drucklos
   ALARM_147 : BOOL ;	//Spannsystem Endlage der Spannvorrichtung nicht erreicht (Drehbewegung Pos.0)
   ALARM_148 : BOOL ;	//Spannsystem Endlage der Spannvorrichtung nicht erreicht (Drehbewegung Pos.1)
   F149 : BOOL ;	//1-
   F150 : BOOL ;	//1-
   F151 : BOOL ;	//1-
   F152 : BOOL ;	//1-
   F153 : BOOL ;	//1-
   F154 : BOOL ;	//1-
   F155 : BOOL ;	//1-
   F156 : BOOL ;	//1-
   F157 : BOOL ;	//1-
   F158 : BOOL ;	//1-
   F159 : BOOL ;	//1-
   F160 : BOOL ;	//1-
   F161 : BOOL ;	//Magnetspannsystem nicht korrekt gespannt /Freigabe PW nicht möglich
   F162 : BOOL ;	//Magnetspannsystem Steckverbindung nicht in Ablagevorrichtung
   F163 : BOOL ;	//1-
   F164 : BOOL ;	//1-
   F165 : BOOL ;	//1-
   F166 : BOOL ;	//1-
   F167 : BOOL ;	//1-
   F168 : BOOL ;	//1-
   F169 : BOOL ;	//1-
   F170 : BOOL ;	//1-
   F171 : BOOL ;	//1-
   F172 : BOOL ;	//1-
   F173 : BOOL ;	//1-
   F174 : BOOL ;	//1-
   F175 : BOOL ;	//1-
   F176 : BOOL ;	//1-
   ALARM_177 : BOOL ;	//min. Füllstand in Behälter MMS unterschritten
   F178 : BOOL ;	//1-
   F179 : BOOL ;	//1-
   F180 : BOOL ;	//1-
   F181 : BOOL ;	//1-
   F182 : BOOL ;	//1-
   F183 : BOOL ;	//1-
   F184 : BOOL ;	//1-
   F185 : BOOL ;	//1-
   F186 : BOOL ;	//1-
   F187 : BOOL ;	//1-
   F188 : BOOL ;	//1-
   F189 : BOOL ;	//1-
   F190 : BOOL ;	//1-
   F191 : BOOL ;	//1-
   F192 : BOOL ;	//1-
   Alarm_193 : BOOL ;	//LUB: Druck an Schmierverteiler Querachse nicht erreicht
   Alarm_194 : BOOL ;	//LUB: Zeitüberschreitung beim Abschalten der Schmierung (Querachse)
   Alarm_195 : BOOL ;	//LUB: Druck an Schmierverteiler Längsachse nicht erreicht
   Alarm_196 : BOOL ;	//LUB: Zeitüberschreitung beim Abschalten der Schmierung (Längsachse)
   Alarm_197 : BOOL ;	//LUB: Druck an Schmierverteiler Vertikalachse nicht erreicht
   Alarm_198 : BOOL ;	//LUB: Zeitüberschreitung beim Abschalten der Schmierung (Vertikalachse)
   Alarm_199 : BOOL ;	//LUB: Druck an Schmierverteiler des Palettenwechsler nicht erreicht
   Alarm_200 : BOOL ;	//LUB: Zeitüberschreitung beim Abschalten der Schmierung (Palettenwechsler)
   Alarm_201 : BOOL ;	//LUB: Druck an Schmierverteiler des Werkzeugmagazin-/wechsler nicht erreicht
   Alarm_202 : BOOL ;	//LUB: Zeitüberschreitung beim Abschalten der Schmierung (Werkzeugmagazin-/wech)
   Alarm_203 : BOOL ;	//LUB: Druck an Schmierverteiler des Rüstplatzes nicht erreicht
   Alarm_204 : BOOL ;	//LUB: Zeitüberschreitung beim Abschalten der Schmierung (Rüstplatzes)
   Alarm_205 : BOOL ;	//LUB: Druck an Schmierverteiler Querachse_1 nicht erreicht
   Alarm_206 : BOOL ;	//LUB: Zeitüberschreitung beim Abschalten der Schmierung (Querachse_1)
   Alarm_207 : BOOL ;	//LUB: Druck an Schmierverteiler Längsachse_1 nicht erreicht
   Alarm_208 : BOOL ;	//LUB: Zeitüberschreitung beim Abschalten der Schmierung (Längsachse_1)
   Alarm_209 : BOOL ;	//LUB: Druck an Schmierverteiler NC-Rundtisch nicht erreicht
   Alarm_210 : BOOL ;	//LUB: Zeitüberschreitung beim Abschalten der Schmierung (NC-Rundtisch)
   F211 : BOOL ;	//1-
   F212 : BOOL ;	//1-
   F213 : BOOL ;	//1-
   F214 : BOOL ;	//1-
   F215 : BOOL ;	//1-
   F216 : BOOL ;	//1-
   F217 : BOOL ;	//1-
   F218 : BOOL ;	//1-
   F219 : BOOL ;	//1-
   F220 : BOOL ;	//1-
   F221 : BOOL ;	//1-
   F222 : BOOL ;	//1-
   F223 : BOOL ;	//1-
   F224 : BOOL ;	//1-
   F225 : BOOL ;	//1-
   F226 : BOOL ;	//1-
   F227 : BOOL ;	//1-
   F228 : BOOL ;	//1-
   F229 : BOOL ;	//1-
   F230 : BOOL ;	//1-
   F231 : BOOL ;	//1-
   F232 : BOOL ;	//1-
   F233 : BOOL ;	//1-
   F234 : BOOL ;	//1-
   F235 : BOOL ;	//1-
   F236 : BOOL ;	//1-
   F237 : BOOL ;	//1-
   F238 : BOOL ;	//1-
   F239 : BOOL ;	//1-
   F240 : BOOL ;	//1-
   F241 : BOOL ;	//1-
   F242 : BOOL ;	//1-
   F243 : BOOL ;	//1-
   F244 : BOOL ;	//1-
   F245 : BOOL ;	//1-
   F246 : BOOL ;	//1-
   F247 : BOOL ;	//1-
   F248 : BOOL ;	//1-
   F249 : BOOL ;	//1-
   F250 : BOOL ;	//1-
   F251 : BOOL ;	//1-
   F252 : BOOL ;	//1-
   F253 : BOOL ;	//1-
   F254 : BOOL ;	//1-
   F255 : BOOL ;	//1-
   F256 : BOOL ;	//1-
   F257 : BOOL ;	//1-
   F258 : BOOL ;	//1-
   F259 : BOOL ;	//1-
   F260 : BOOL ;	//1-
   F261 : BOOL ;	//1-
   F262 : BOOL ;	//1-
   F263 : BOOL ;	//1-
   F264 : BOOL ;	//1-
   F265 : BOOL ;	//1-
   F266 : BOOL ;	//1-
   F267 : BOOL ;	//1-
   F268 : BOOL ;	//1-
   F269 : BOOL ;	//1-
   F270 : BOOL ;	//1-
   F271 : BOOL ;	//1-
   F272 : BOOL ;	//1-
   F273 : BOOL ;	//1-
   F274 : BOOL ;	//1-
   F275 : BOOL ;	//1-
   F276 : BOOL ;	//1-
   F277 : BOOL ;	//1-
   F278 : BOOL ;	//1-
   F279 : BOOL ;	//1-
   F280 : BOOL ;	//1-
   F281 : BOOL ;	//1-
   F282 : BOOL ;	//1-
   F283 : BOOL ;	//1-
   F284 : BOOL ;	//1-
   F285 : BOOL ;	//1-
   F286 : BOOL ;	//1-
   F287 : BOOL ;	//1-
   F288 : BOOL ;	//1-
   F289 : BOOL ;	//1-
   F290 : BOOL ;	//1-
   F291 : BOOL ;	//1-
   F292 : BOOL ;	//1-
   F293 : BOOL ;	//1-
   F294 : BOOL ;	//1-
   F295 : BOOL ;	//1-
   F296 : BOOL ;	//1-
   F297 : BOOL ;	//1-
   F298 : BOOL ;	//1-
   F299 : BOOL ;	//1-
   F300 : BOOL ;	//1-
   F301 : BOOL ;	//1-
   F302 : BOOL ;	//1-
   F303 : BOOL ;	//1-
   F304 : BOOL ;	//1-
   F305 : BOOL ;	//1-
   F306 : BOOL ;	//1-
   F307 : BOOL ;	//1-
   F308 : BOOL ;	//1-
   F309 : BOOL ;	//1-
   F310 : BOOL ;	//1-
   F311 : BOOL ;	//1-
   F312 : BOOL ;	//1-
   F313 : BOOL ;	//1-
   F314 : BOOL ;	//1-
   F315 : BOOL ;	//1-
   F316 : BOOL ;	//1-
   F317 : BOOL ;	//1-
   F318 : BOOL ;	//1-
   F319 : BOOL ;	//1-
   F320 : BOOL ;	//1-
   F321 : BOOL ;	//1-
   F322 : BOOL ;	//1-
   F323 : BOOL ;	//1-
   F324 : BOOL ;	//1-
   F325 : BOOL ;	//1-
   F326 : BOOL ;	//1-
   F327 : BOOL ;	//1-
   F328 : BOOL ;	//1-
   F329 : BOOL ;	//1-
   F330 : BOOL ;	//1-
   F331 : BOOL ;	//1-
   F332 : BOOL ;	//1-
   F333 : BOOL ;	//1-
   F334 : BOOL ;	//1-
   F335 : BOOL ;	//1-
   F336 : BOOL ;	//1-
   F337 : BOOL ;	//1-
   F338 : BOOL ;	//1-
   F339 : BOOL ;	//1-
   F340 : BOOL ;	//1-
   F341 : BOOL ;	//1-
   F342 : BOOL ;	//1-
   F343 : BOOL ;	//1-
   F344 : BOOL ;	//1-
   F345 : BOOL ;	//1-
   F346 : BOOL ;	//1-
   F347 : BOOL ;	//1-
   F348 : BOOL ;	//1-
   F349 : BOOL ;	//1-
   F350 : BOOL ;	//1-
   F351 : BOOL ;	//1-
   F352 : BOOL ;	//1-
   F353 : BOOL ;	//1-
   F354 : BOOL ;	//1-
   F355 : BOOL ;	//1-
   F356 : BOOL ;	//1-
   F357 : BOOL ;	//1-
   F358 : BOOL ;	//1-
   F359 : BOOL ;	//1-
   F360 : BOOL ;	//1-
   F361 : BOOL ;	//1-
   F362 : BOOL ;	//1-
   F363 : BOOL ;	//1-
   F364 : BOOL ;	//1-
   F365 : BOOL ;	//1-
   F366 : BOOL ;	//1-
   F367 : BOOL ;	//1-
   F368 : BOOL ;	//1-
   F369 : BOOL ;	//1-
   F370 : BOOL ;	//1-
   F371 : BOOL ;	//1-
   F372 : BOOL ;	//1-
   F373 : BOOL ;	//1-
   F374 : BOOL ;	//1-
   F375 : BOOL ;	//1-
   F376 : BOOL ;	//1-
   F377 : BOOL ;	//1-
   F378 : BOOL ;	//1-
   F379 : BOOL ;	//1-
   F380 : BOOL ;	//1-
   F381 : BOOL ;	//1-
   F382 : BOOL ;	//1-
   F383 : BOOL ;	//1-
   F384 : BOOL ;	//1-
   F385 : BOOL ;	//1-
   F386 : BOOL ;	//1-
   F387 : BOOL ;	//1-
   F388 : BOOL ;	//1-
   F389 : BOOL ;	//1-
   F390 : BOOL ;	//1-
   F391 : BOOL ;	//1-
   F392 : BOOL ;	//1-
   F393 : BOOL ;	//1-
   F394 : BOOL ;	//1-
   F395 : BOOL ;	//1-
   F396 : BOOL ;	//1-
   F397 : BOOL ;	//1-
   F398 : BOOL ;	//1-
   F399 : BOOL ;	//1-
   F400 : BOOL ;	//1-
   F401 : BOOL ;	//1-
   F402 : BOOL ;	//1-
   F403 : BOOL ;	//1-
   F404 : BOOL ;	//1-
   F405 : BOOL ;	//1-
   F406 : BOOL ;	//1-
   F407 : BOOL ;	//1-
   F408 : BOOL ;	//1-
   F409 : BOOL ;	//1-
   F410 : BOOL ;	//1-
   F411 : BOOL ;	//1-
   F412 : BOOL ;	//1-
   F413 : BOOL ;	//1-
   F414 : BOOL ;	//1-
   F415 : BOOL ;	//1-
   F416 : BOOL ;	//1-
   F417 : BOOL ;	//1-
   F418 : BOOL ;	//1-
   F419 : BOOL ;	//1-
   F420 : BOOL ;	//1-
   F421 : BOOL ;	//1-
   F422 : BOOL ;	//1-
   F423 : BOOL ;	//1-
   F424 : BOOL ;	//1-
   F425 : BOOL ;	//1-
   F426 : BOOL ;	//1-
   F427 : BOOL ;	//1-
   F428 : BOOL ;	//1-
   F429 : BOOL ;	//1-
   F430 : BOOL ;	//1-
   F431 : BOOL ;	//1-
   F432 : BOOL ;	//1-
   F433 : BOOL ;	//1-
   F434 : BOOL ;	//1-
   F435 : BOOL ;	//1-
   F436 : BOOL ;	//1-
   F437 : BOOL ;	//1-
   F438 : BOOL ;	//1-
   F439 : BOOL ;	//1-
   F440 : BOOL ;	//1-
   F441 : BOOL ;	//1-
   F442 : BOOL ;	//1-
   F443 : BOOL ;	//1-
   F444 : BOOL ;	//1-
   F445 : BOOL ;	//1-
   F446 : BOOL ;	//1-
   F447 : BOOL ;	//1-
   F448 : BOOL ;	//1-
   F449 : BOOL ;	//1-
   F450 : BOOL ;	//1-
   F451 : BOOL ;	//1-
   F452 : BOOL ;	//1-
   F453 : BOOL ;	//1-
   F454 : BOOL ;	//1-
   F455 : BOOL ;	//1-
   F456 : BOOL ;	//1-
   F457 : BOOL ;	//1-
   F458 : BOOL ;	//1-
   F459 : BOOL ;	//1-
   F460 : BOOL ;	//1-
   F461 : BOOL ;	//1-
   F462 : BOOL ;	//1-
   F463 : BOOL ;	//1-
   F464 : BOOL ;	//1-
   F465 : BOOL ;	//1-
   F466 : BOOL ;	//1-
   F467 : BOOL ;	//1-
   F468 : BOOL ;	//1-
   F469 : BOOL ;	//1-
   F470 : BOOL ;	//1-
   F471 : BOOL ;	//1-
   F472 : BOOL ;	//1-
   F473 : BOOL ;	//1-
   F474 : BOOL ;	//1-
   F475 : BOOL ;	//1-
   F476 : BOOL ;	//1-
   F477 : BOOL ;	//1-
   F478 : BOOL ;	//1-
   F479 : BOOL ;	//1-
   F480 : BOOL ;	//1-
   F481 : BOOL ;	//1-
   F482 : BOOL ;	//1-
   F483 : BOOL ;	//1-
   F484 : BOOL ;	//1-
   F485 : BOOL ;	//1-
   F486 : BOOL ;	//1-
   F487 : BOOL ;	//1-
   F488 : BOOL ;	//1-
   F489 : BOOL ;	//1-
   F490 : BOOL ;	//1-
   F491 : BOOL ;	//1-
   F492 : BOOL ;	//1-
   F493 : BOOL ;	//1-
   F494 : BOOL ;	//1-
   F495 : BOOL ;	//1-
   F496 : BOOL ;	//1-
   F497 : BOOL ;	//1-
   F498 : BOOL ;	//1-
   F499 : BOOL ;	//1-
   F500 : BOOL ;	//1-
   F501 : BOOL ;	//1-
   F502 : BOOL ;	//1-
   F503 : BOOL ;	//1-
   F504 : BOOL ;	//1-
   F505 : BOOL ;	//1-
   F506 : BOOL ;	//1-
   F507 : BOOL ;	//1-
   F508 : BOOL ;	//1-
   F509 : BOOL ;	//1-
   F510 : BOOL ;	//1-
   F511 : BOOL ;	//1-
   F512 : BOOL ;	//1-
   MSG_513 : BOOL ;	//Schaltschranktüre(n) an Werkzeugmaschine geöffnet
   MSG_514 : BOOL ;	//Schaltschranktüre(n) an Kühlschmierstoffanlage geöffnet
   MSG_515 : BOOL ;	//Schaltschranktemperatur zu hoch
   Me516 : BOOL ;	//1-
   Me517 : BOOL ;	//1-
   Me518 : BOOL ;	//1-
   Me519 : BOOL ;	//1-
   Me520 : BOOL ;	//1-
   Me521 : BOOL ;	//1-
   Me522 : BOOL ;	//1-
   Me523 : BOOL ;	//1-
   Me524 : BOOL ;	//1-
   Me525 : BOOL ;	//1-
   Me526 : BOOL ;	//1-
   Me527 : BOOL ;	//1-
   Me528 : BOOL ;	//1-
   MSG_529 : BOOL ;	//Hydraulikfilter Maschine verschmutzt
   MSG_530 : BOOL ;	//HYD:Hydraulik Maschine Füllstand Maximum überschritten
   MSG_531 : BOOL ;	//HYD:Hydraulik Maschine Füllstand Minimum unterschritten
   Me532 : BOOL ;	//1-
   Me533 : BOOL ;	//1-
   Me534 : BOOL ;	//1-
   Me535 : BOOL ;	//1-
   Me536 : BOOL ;	//1-
   Me537 : BOOL ;	//1-
   Me538 : BOOL ;	//1-
   Me539 : BOOL ;	//1-
   Me540 : BOOL ;	//1-
   Me541 : BOOL ;	//1-
   Me542 : BOOL ;	//1-
   Me543 : BOOL ;	//1-
   Me544 : BOOL ;	//1-
   MSG_545 : BOOL ;	//Vakuumspannsystem nicht gespannt (Arbeitsraum)
   MSG_546 : BOOL ;	//Vakuumspannsystem nicht gespannt (Rüstplatz)
   MSG_547 : BOOL ;	//Vakuumspannsystem: Lösen nicht möglich
   Me548 : BOOL ;	//1-
   Me549 : BOOL ;	//1-
   Me550 : BOOL ;	//1-
   Me551 : BOOL ;	//1-
   Me552 : BOOL ;	//1-
   Me553 : BOOL ;	//1-
   Me554 : BOOL ;	//1-
   Me555 : BOOL ;	//1-
   Me556 : BOOL ;	//1-
   Me557 : BOOL ;	//1-
   Me558 : BOOL ;	//1-
   Me559 : BOOL ;	//1-
   Me560 : BOOL ;	//1-
   MSG_561 : BOOL ;	//Warnung von Kühlschmierstoffanlage
   MSG_562 : BOOL ;	//Warnung! Feinfilter Kühlschmierstoffanlage verschmutzt
   MSG_563 : BOOL ;	//Die gewählte Druckstufe liegt nicht im möglichen Wertebereich!
   Me564 : BOOL ;	//1-
   Me565 : BOOL ;	//1-
   Me566 : BOOL ;	//1-
   Me567 : BOOL ;	//1-
   Me568 : BOOL ;	//1-
   Me569 : BOOL ;	//1-
   Me570 : BOOL ;	//1-
   Me571 : BOOL ;	//1-
   Me572 : BOOL ;	//1-
   Me573 : BOOL ;	//1-
   Me574 : BOOL ;	//1-
   Me575 : BOOL ;	//1-
   Me576 : BOOL ;	//1-
   MSG_577 : BOOL ;	//Löseanforderung von extern aber keine Freigabe von LeitPLC
   MSG_578 : BOOL ;	//Löseanforderung aber Spannsystem nicht aktiviert
   MSG_579 : BOOL ;	//Nullpunktspannsstem ist gelöst
   Me580 : BOOL ;	//1-
   Me581 : BOOL ;	//1-
   Me582 : BOOL ;	//1-
   Me583 : BOOL ;	//1-
   Me584 : BOOL ;	//1-
   Me585 : BOOL ;	//1-
   Me586 : BOOL ;	//1-
   Me587 : BOOL ;	//1-
   Me588 : BOOL ;	//1-
   Me589 : BOOL ;	//1-
   Me590 : BOOL ;	//1-
   Me591 : BOOL ;	//1-
   Me592 : BOOL ;	//1-
   MSG_593 : BOOL ;	//Vorwarnung min. Füllstand Behälter MMS
   MSG_594 : BOOL ;	//min.Füllstand in Versorgungseinheit MMS unterschritten
   Me595 : BOOL ;	//1-
   Me596 : BOOL ;	//1-
   Me597 : BOOL ;	//1-
   Me598 : BOOL ;	//1-
   Me599 : BOOL ;	//1-
   MSG_600 : BOOL ;	//NOT-AUS Bedienpult betätigt
   MSG_601 : BOOL ;	//NOT-AUS Bedienpult Handrad betätigt
   MSG_602 : BOOL ;	//NOT-AUS Späneförderer betätigt
   MSG_603 : BOOL ;	//NOT-AUS Werkzeugeingabestation betätigt
   MSG_604 : BOOL ;	//NOT-AUS Rüstplatz betätigt
   MSG_605 : BOOL ;	//NOT-AUS Werkzeugmagazin Handrad betätigt
   MSG_606 : BOOL ;	//NOT-Aus Werkzeugmagazin
   Me607 : BOOL ;	//1-
   Me608 : BOOL ;	//1-
   Me609 : BOOL ;	//1-
   Me610 : BOOL ;	//1-
   MSG_611 : BOOL ;	//Leitungsschutzschalter Steckdose Frontschild hat ausgelöst
   MSG_612 : BOOL ;	//Leitungsschutzschalter Schmierstoffpumpe hat ausgelöst
   MSG_613 : BOOL ;	//Leitungsschutzschalter AS-i Netzteil hat ausgelöst
   MSG_614 : BOOL ;	//Leitungsschutzschalter Durchflussüberwachung hat ausgelöst
   MSG_615 : BOOL ;	//Leitungsschutzschalter Leuchtmelder Kommandostation hat ausgelöst
   MSG_616 : BOOL ;	//Leitungsschutzschalter Steuerstromkreis hat ausgelöst
   MSG_617 : BOOL ;	//Leitungsschutzschalter CNC-Steuerung hat ausgelöst
   MSG_618 : BOOL ;	//Leitungsschutzschalter Not-Aus Steuerstromkreis hat ausgelöst
   MSG_619 : BOOL ;	//Leitungsschutzschalter Werkzeugwechsler hat ausgelöst
   MSG_620 : BOOL ;	//Leitungsschutzschalter DC-Steuerspannung hat ausgelöst
   MSG_621 : BOOL ;	//Leitungsschutzschalter Palettenwechsler hat ausgelöst
   MSG_622 : BOOL ;	//Leitungsschutzschalter Kühlmittelanlage hat ausgelöst
   MSG_623 : BOOL ;	//Leitungsschutzschalter PCU 50 hat ausgelöst
   MSG_624 : BOOL ;	//Leitungsschutzschalter Bildschirm hat ausgelöst
   MSG_625 : BOOL ;	//Leitungsschutzschalter IM151 Maschine hat ausgelöst
   MSG_626 : BOOL ;	//Leitungsschutzschalter_1 Ausgänge IM151 hat ausgelöst
   MSG_627 : BOOL ;	//Leitungsschutzschalter_2 Ausgänge IM151 hat ausgelöst
   MSG_628 : BOOL ;	//Leitungsschutzschalter Drehzahl Überwachung hat ausgelöst
   MSG_629 : BOOL ;	//Leitungsschutzschalter Netzteil Werkzeugwechsler hat ausgelöst
   MSG_630 : BOOL ;	//Leitungsschutzschalter Werkzeugidentifikation hat ausgelöst
   MSG_631 : BOOL ;	//Leitungsschutzschalter Werkzeugkegelreinigung hat ausgelöst
   MSG_632 : BOOL ;	//Leitungsschutzschalter Steuerstromkreis Palettenspeiche/-wechsler hat ausgelöst
   MSG_633 : BOOL ;	//Leitungsschutzschalter Bremse Palettenspeicher/-wechsler hat ausgelöst
   MSG_634 : BOOL ;	//Leitungsschutzschalter Betriebsdatenerfassung hat ausgelöst
   MSG_635 : BOOL ;	//Leitungsschutzschalter Werkzeugbruchüberwachung hat ausgelöst
   MSG_636 : BOOL ;	//Leitungsschutzschalter Minimalmengenschmierung hat ausgelöst
   MSG_637 : BOOL ;	//Leitungsschutzschalter Tuning IM 151_4 hat ausgelöst
   MSG_638 : BOOL ;	//Leitungsschutzschalter Tuning Ausgänge IM 151 hat ausgelöst
   MSG_639 : BOOL ;	//Leitungsschutzschalter Tuning Eingänge IM 151 hat ausgelöst
   MSG_640 : BOOL ;	//Leitungsschutzschalter Schaltschrankbeleuchtung hat ausgelöst
   MSG_641 : BOOL ;	//Leitungsschutzschalter Tuning IM 151_7 hat ausgelöst
   MSG_642 : BOOL ;	//Leitungsschutzschalter Drehzahl Überwachung Rüstplatz hat ausgelöst
   MSG_643 : BOOL ;	//Leitungsschutzschalter Messtaster hat ausgelöst
   MSG_644 : BOOL ;	//Leitungsschutzschalter Kabinentüre hat ausgelöst
   MSG_645 : BOOL ;	//Leitungsschutzschalter Leistung Spindel hat ausgelöst
   MSG_646 : BOOL ;	//Leitungsschutzschalter 230V hat ausgelöst
   MSG_647 : BOOL ;	//Leitungsschutzschalter 24V hat ausgelöst
   Me648 : BOOL ;	//1-
   Me649 : BOOL ;	//1-
   MSG_650 : BOOL ;	//TMS: Leitungsschutzschalter Bremse hat ausgelöst
   MSG_651 : BOOL ;	//TMS: Leitungsschutzschalter AC-Steuerspannung hat ausgelöst
   MSG_652 : BOOL ;	//TMS: Leitungsschutzschalter Steuerstromkreis hat ausgelöst
   MSG_653 : BOOL ;	//TMS: Leitungsschutzschalter Werkzeugeingabestation hat ausgelöst
   MSG_654 : BOOL ;	//TMS: Leitungsschutzschalter Ausgänge hat ausgelöst
   MSG_655 : BOOL ;	//TMS: Leitungsschutzschalter Netzteil hat ausgelöst
   Me656 : BOOL ;	//1-
   Me657 : BOOL ;	//1-
   MSG_658 : BOOL ;	//KSA: Leitungsschutzschalter Sensoren hat ausgelöst
   MSG_659 : BOOL ;	//KSA: Leitungsschutzschalter Proportionalventil 1 hat ausgelöst
   MSG_660 : BOOL ;	//KSA: Leitungsschutzschalter Proportionalventil 2 hat ausgelöst
   Me661 : BOOL ;	//1-
   Me662 : BOOL ;	//1-
   Me663 : BOOL ;	//1-
   Me664 : BOOL ;	//1-
   Me665 : BOOL ;	//1-
   Me666 : BOOL ;	//1-
   Me667 : BOOL ;	//1-
   Me668 : BOOL ;	//1-
   Me669 : BOOL ;	//1-
   Me670 : BOOL ;	//1-
   Me671 : BOOL ;	//1-
   Me672 : BOOL ;	//1-
   Me673 : BOOL ;	//1-
   Me674 : BOOL ;	//1-
   Me675 : BOOL ;	//1-
   MSG_676 : BOOL ;	//Leistungsschalter Späneförderer 2 hat ausgelöst
   MSG_677 : BOOL ;	//Leistungsschalter Kabinentüre hat ausgelöst
   MSG_678 : BOOL ;	//Leistungsschalter Steckdose Bedienpult hat ausgelöst
   MSG_679 : BOOL ;	//Leistungsschalter Steckdose Palettenwechsler hat ausgelöst
   MSG_680 : BOOL ;	//Leistungsschalter Schaltschrankbeleuchtung hat ausgelöst
   MSG_681 : BOOL ;	//Leistungsschalter DC-Steuerspannung_1 hat ausgelöst
   MSG_682 : BOOL ;	//Leistungsschalter DC-Steuerspannung_2 hat ausgelöst
   MSG_683 : BOOL ;	//Leistungsschalter AC-Steurspannung hat ausgelöst
   MSG_684 : BOOL ;	//Leistungsschalter Kühl-/Heizaggregat hat ausgelöst
   MSG_685 : BOOL ;	//Leistungsschalter AC-Versorgungsmodul hat ausgelöst
   MSG_686 : BOOL ;	//Leistungsschalter Lüfter AC hat ausgelöst
   MSG_687 : BOOL ;	//Leistungsschalter Kühlaggregat Schaltschrank hat ausgelöst
   MSG_688 : BOOL ;	//Leistungsschalter Werkzeugregal hat ausgelöst
   MSG_689 : BOOL ;	//Leistungsschalter Lüfter FD hat ausgelöst
   MSG_690 : BOOL ;	//Leistungsschalter Kühlmittelanlage hat ausgelöst
   Me691 : BOOL ;	//1-
   Me692 : BOOL ;	//1-
   MSG_693 : BOOL ;	//TMS: Leistungsschalter AC-Steuerspannung hat ausgelöst
   MSG_694 : BOOL ;	//TMS: Leistungsschalter Antriebe hat ausgelöst
   Me695 : BOOL ;	//1-
   Me696 : BOOL ;	//1-
   Me697 : BOOL ;	//1-
   Me698 : BOOL ;	//1-
   Me699 : BOOL ;	//1-
   MSG_700 : BOOL ;	//KSA: Leistungsschalter Pumpe Spänespülung Dach hat ausgelöst
   MSG_701 : BOOL ;	//KSA: Leistungsschalter Pumpe Spülpistole hat ausgelöst
   MSG_702 : BOOL ;	//KSA: Leistungsschalter Pumpe Spänespülung Türe hat ausgelöst
   MSG_703 : BOOL ;	//KSA: Leistungsschalter Pumpe Feinstbereich hat ausgelöst
   MSG_704 : BOOL ;	//KSA: Leistungsschalter Kratzerförder hat ausgelöst
   MSG_705 : BOOL ;	//KSA: Leistungsschalter Pumpe Kühlmittel 1 hat ausgelöst
   MSG_706 : BOOL ;	//KSA: Hauptschalter Kühlmittelanlage hat ausgelöst
   MSG_707 : BOOL ;	//KSA: Leistungsschalter Pumpe 40b hat ausgelöst
   MSG_708 : BOOL ;	//KSA: Leistungsschalter Pumpe 80b hat ausgelöst
   Me709 : BOOL ;	//1-
   Me710 : BOOL ;	//1-
   Me711 : BOOL ;	//1-
   Me712 : BOOL ;	//1-
   Me713 : BOOL ;	//1-
   Me714 : BOOL ;	//1-
   MSG_715 : BOOL ;	//KSA-Temp: Leistungsschalter Kompressor hat ausgelöst
   MSG_716 : BOOL ;	//KSA-Temp: Leistungsschalter Lüfter hat ausgelöst
   MSG_717 : BOOL ;	//KSA-Temp: Leistungsschalter Rührwerk hat ausgelöst
   MSG_718 : BOOL ;	//KSA-Temp: Leistungsschalter Hebepumpe hat ausgelöst
   MSG_719 : BOOL ;	//KSA-Temp: Leistungsschalter Heizung hat ausgelöst
   MSG_720 : BOOL ;	//KSA-Temp: Leistungsschalter Steuerspannung hat ausgelöst
   Me721 : BOOL ;	//1-
   Me722 : BOOL ;	//1-
   Me723 : BOOL ;	//1-
   Me724 : BOOL ;	//1-
   MSG_725 : BOOL ;	//Wartungstüre Werkzeugmagazin ist offen
   MSG_726 : BOOL ;	//Wartungstüre Werkzeugregal ist offen
   MSG_727 : BOOL ;	//Wartungstüre Werkzeugeingabestation ist offen
   MSG_728 : BOOL ;	//Wartungstüre Palettenspeicher/-wechsler ist offen
   Me729 : BOOL ;	//1-
   Me730 : BOOL ;	//1-
   Me731 : BOOL ;	//1-
   Me732 : BOOL ;	//1-
   Me733 : BOOL ;	//1-
   Me734 : BOOL ;	//1-
   Me735 : BOOL ;	//1-
   Me736 : BOOL ;	//1-
   Me737 : BOOL ;	//1-
   Me738 : BOOL ;	//1-
   Me739 : BOOL ;	//1-
   Me740 : BOOL ;	//1-
   Me741 : BOOL ;	//1-
   Me742 : BOOL ;	//1-
   Me743 : BOOL ;	//1-
   Me744 : BOOL ;	//1-
   Me745 : BOOL ;	//1-
   Me746 : BOOL ;	//1-
   Me747 : BOOL ;	//1-
   Me748 : BOOL ;	//1-
   Me749 : BOOL ;	//1-
   Me750 : BOOL ;	//1-
   Me751 : BOOL ;	//1-
   Me752 : BOOL ;	//1-
   Me753 : BOOL ;	//1-
   Me754 : BOOL ;	//1-
   Me755 : BOOL ;	//1-
   Me756 : BOOL ;	//1-
   Me757 : BOOL ;	//1-
   Me758 : BOOL ;	//1-
   Me759 : BOOL ;	//1-
   Me760 : BOOL ;	//1-
   Me761 : BOOL ;	//1-
   Me762 : BOOL ;	//1-
   Me763 : BOOL ;	//1-
   Me764 : BOOL ;	//1-
   Me765 : BOOL ;	//1-
   Me766 : BOOL ;	//1-
   Me767 : BOOL ;	//1-
   Me768 : BOOL ;	//1-
   Me769 : BOOL ;	//1-
   Me770 : BOOL ;	//1-
   Me771 : BOOL ;	//1-
   Me772 : BOOL ;	//1-
   Me773 : BOOL ;	//1-
   Me774 : BOOL ;	//1-
   Me775 : BOOL ;	//1-
   Me776 : BOOL ;	//1-
   Me777 : BOOL ;	//1-
   Me778 : BOOL ;	//1-
   Me779 : BOOL ;	//1-
   Me780 : BOOL ;	//1-
   Me781 : BOOL ;	//1-
   Me782 : BOOL ;	//1-
   Me783 : BOOL ;	//1-
   Me784 : BOOL ;	//1-
   Me785 : BOOL ;	//1-
   Me786 : BOOL ;	//1-
   Me787 : BOOL ;	//1-
   Me788 : BOOL ;	//1-
   Me789 : BOOL ;	//1-
   Me790 : BOOL ;	//1-
   Me791 : BOOL ;	//1-
   Me792 : BOOL ;	//1-
   Me793 : BOOL ;	//1-
   Me794 : BOOL ;	//1-
   Me795 : BOOL ;	//1-
   Me796 : BOOL ;	//1-
   Me797 : BOOL ;	//1-
   Me798 : BOOL ;	//1-
   Me799 : BOOL ;	//1-
   Me800 : BOOL ;	//1-
   Me801 : BOOL ;	//1-
   Me802 : BOOL ;	//1-
   Me803 : BOOL ;	//1-
   Me804 : BOOL ;	//1-
   Me805 : BOOL ;	//1-
   Me806 : BOOL ;	//1-
   Me807 : BOOL ;	//1-
   Me808 : BOOL ;	//1-
   Me809 : BOOL ;	//1-
   Me810 : BOOL ;	//1-
   Me811 : BOOL ;	//1-
   Me812 : BOOL ;	//1-
   Me813 : BOOL ;	//1-
   Me814 : BOOL ;	//1-
   Me815 : BOOL ;	//1-
   Me816 : BOOL ;	//1-
   Me817 : BOOL ;	//1-
   Me818 : BOOL ;	//1-
   Me819 : BOOL ;	//1-
   Me820 : BOOL ;	//1-
   Me821 : BOOL ;	//1-
   Me822 : BOOL ;	//1-
   Me823 : BOOL ;	//1-
   Me824 : BOOL ;	//1-
   Me825 : BOOL ;	//1-
   Me826 : BOOL ;	//1-
   Me827 : BOOL ;	//1-
   Me828 : BOOL ;	//1-
   Me829 : BOOL ;	//1-
   Me830 : BOOL ;	//1-
   Me831 : BOOL ;	//1-
   Me832 : BOOL ;	//1-
   Me833 : BOOL ;	//1-
   Me834 : BOOL ;	//1-
   Me835 : BOOL ;	//1-
   Me836 : BOOL ;	//1-
   Me837 : BOOL ;	//1-
   Me838 : BOOL ;	//1-
   Me839 : BOOL ;	//1-
   Me840 : BOOL ;	//1-
   Me841 : BOOL ;	//1-
   Me842 : BOOL ;	//1-
   Me843 : BOOL ;	//1-
   Me844 : BOOL ;	//1-
   Me845 : BOOL ;	//1-
   Me846 : BOOL ;	//1-
   Me847 : BOOL ;	//1-
   Me848 : BOOL ;	//1-
   Me849 : BOOL ;	//1-
   Me850 : BOOL ;	//1-
   Me851 : BOOL ;	//1-
   Me852 : BOOL ;	//1-
   Me853 : BOOL ;	//1-
   Me854 : BOOL ;	//1-
   Me855 : BOOL ;	//1-
   Me856 : BOOL ;	//1-
   Me857 : BOOL ;	//1-
   Me858 : BOOL ;	//1-
   Me859 : BOOL ;	//1-
   Me860 : BOOL ;	//1-
   Me861 : BOOL ;	//1-
   Me862 : BOOL ;	//1-
   Me863 : BOOL ;	//1-
   Me864 : BOOL ;	//1-
   Me865 : BOOL ;	//1-
   Me866 : BOOL ;	//1-
   Me867 : BOOL ;	//1-
   Me868 : BOOL ;	//1-
   Me869 : BOOL ;	//1-
   Me870 : BOOL ;	//1-
   Me871 : BOOL ;	//1-
   Me872 : BOOL ;	//1-
   Me873 : BOOL ;	//1-
   Me874 : BOOL ;	//1-
   Me875 : BOOL ;	//1-
   Me876 : BOOL ;	//1-
   Me877 : BOOL ;	//1-
   Me878 : BOOL ;	//1-
   Me879 : BOOL ;	//1-
   Me880 : BOOL ;	//1-
   Me881 : BOOL ;	//1-
   Me882 : BOOL ;	//1-
   Me883 : BOOL ;	//1-
   Me884 : BOOL ;	//1-
   Me885 : BOOL ;	//1-
   Me886 : BOOL ;	//1-
   Me887 : BOOL ;	//1-
   Me888 : BOOL ;	//1-
   Me889 : BOOL ;	//1-
   Me890 : BOOL ;	//1-
   Me891 : BOOL ;	//1-
   Me892 : BOOL ;	//1-
   Me893 : BOOL ;	//1-
   Me894 : BOOL ;	//1-
   Me895 : BOOL ;	//1-
   Me896 : BOOL ;	//1-
   Me897 : BOOL ;	//1-
   Me898 : BOOL ;	//1-
   Me899 : BOOL ;	//1-
   Me900 : BOOL ;	//1-
   Me901 : BOOL ;	//1-
   Me902 : BOOL ;	//1-
   Me903 : BOOL ;	//1-
   Me904 : BOOL ;	//1-
   Me905 : BOOL ;	//1-
   Me906 : BOOL ;	//1-
   Me907 : BOOL ;	//1-
   Me908 : BOOL ;	//1-
   Me909 : BOOL ;	//1-
   Me910 : BOOL ;	//1-
   Me911 : BOOL ;	//1-
   Me912 : BOOL ;	//1-
   Me913 : BOOL ;	//1-
   Me914 : BOOL ;	//1-
   Me915 : BOOL ;	//1-
   Me916 : BOOL ;	//1-
   Me917 : BOOL ;	//1-
   Me918 : BOOL ;	//1-
   Me919 : BOOL ;	//1-
   Me920 : BOOL ;	//1-
   Me921 : BOOL ;	//1-
   Me922 : BOOL ;	//1-
   Me923 : BOOL ;	//1-
   Me924 : BOOL ;	//1-
   Me925 : BOOL ;	//1-
   Me926 : BOOL ;	//1-
   Me927 : BOOL ;	//1-
   Me928 : BOOL ;	//1-
   Me929 : BOOL ;	//1-
   Me930 : BOOL ;	//1-
   Me931 : BOOL ;	//1-
   Me932 : BOOL ;	//1-
   Me933 : BOOL ;	//1-
   Me934 : BOOL ;	//1-
   Me935 : BOOL ;	//1-
   Me936 : BOOL ;	//1-
   Me937 : BOOL ;	//1-
   Me938 : BOOL ;	//1-
   Me939 : BOOL ;	//1-
   Me940 : BOOL ;	//1-
   Me941 : BOOL ;	//1-
   Me942 : BOOL ;	//1-
   Me943 : BOOL ;	//1-
   Me944 : BOOL ;	//1-
   Me945 : BOOL ;	//1-
   Me946 : BOOL ;	//1-
   Me947 : BOOL ;	//1-
   Me948 : BOOL ;	//1-
   Me949 : BOOL ;	//1-
   Me950 : BOOL ;	//1-
   Me951 : BOOL ;	//1-
   Me952 : BOOL ;	//1-
   Me953 : BOOL ;	//1-
   Me954 : BOOL ;	//1-
   Me955 : BOOL ;	//1-
   Me956 : BOOL ;	//1-
   Me957 : BOOL ;	//1-
   Me958 : BOOL ;	//1-
   Me959 : BOOL ;	//1-
   Me960 : BOOL ;	//1-
   Me961 : BOOL ;	//1-
   Me962 : BOOL ;	//1-
   Me963 : BOOL ;	//1-
   Me964 : BOOL ;	//1-
   Me965 : BOOL ;	//1-
   Me966 : BOOL ;	//1-
   Me967 : BOOL ;	//1-
   Me968 : BOOL ;	//1-
   Me969 : BOOL ;	//1-
   Me970 : BOOL ;	//1-
   Me971 : BOOL ;	//1-
   Me972 : BOOL ;	//1-
   Me973 : BOOL ;	//1-
   Me974 : BOOL ;	//1-
   Me975 : BOOL ;	//1-
   Me976 : BOOL ;	//1-
   Me977 : BOOL ;	//1-
   Me978 : BOOL ;	//1-
   Me979 : BOOL ;	//1-
   Me980 : BOOL ;	//1-
   Me981 : BOOL ;	//1-
   Me982 : BOOL ;	//1-
   Me983 : BOOL ;	//1-
   Me984 : BOOL ;	//1-
   Me985 : BOOL ;	//1-
   Me986 : BOOL ;	//1-
   Me987 : BOOL ;	//1-
   Me988 : BOOL ;	//1-
   Me989 : BOOL ;	//1-
   Me990 : BOOL ;	//1-
   Me991 : BOOL ;	//1-
   Me992 : BOOL ;	//1-
   Me993 : BOOL ;	//1-
   Me994 : BOOL ;	//1-
   Me995 : BOOL ;	//1-
   Me996 : BOOL ;	//1-
   Me997 : BOOL ;	//1-
   Me998 : BOOL ;	//1-
   Me999 : BOOL ;	//1-
   Me1000 : BOOL ;	//1-
   Me1001 : BOOL ;	//1-
   Me1002 : BOOL ;	//1-
   Me1003 : BOOL ;	//1-
   Me1004 : BOOL ;	//1-
   Me1005 : BOOL ;	//1-
   Me1006 : BOOL ;	//1-
   Me1007 : BOOL ;	//1-
   Me1008 : BOOL ;	//1-
   Me1009 : BOOL ;	//1-
   Me1010 : BOOL ;	//1-
   Me1011 : BOOL ;	//1-
   Me1012 : BOOL ;	//1-
   Me1013 : BOOL ;	//1-
   Me1014 : BOOL ;	//1-
   Me1015 : BOOL ;	//1-
   Me1016 : BOOL ;	//1-
   Me1017 : BOOL ;	//1-
   Me1018 : BOOL ;	//1-
   Me1019 : BOOL ;	//1-
   Me1020 : BOOL ;	//1-
   Me1021 : BOOL ;	//1-
   Me1022 : BOOL ;	//1-
   Me1023 : BOOL ;	//1-
   Me1024 : BOOL ;	//1-
  END_STRUCT ;	
BEGIN
END_DATA_BLOCK

DATA_BLOCK DB 20
AUTHOR : SPAC_slh
FAMILY : AUTOMAT
VERSION : 0.0
"AutoSusDoor"
BEGIN
END_DATA_BLOCK

DATA_BLOCK "INS_MESSAGE_OUT"	// DB 100
AUTHOR : SPAC_slh
VERSION : 0.0
"MESSAGE_OUT"
BEGIN
END_DATA_BLOCK

DATA_BLOCK "DB_CK_OP"	// DB 101
VERSION : 0.1
  STRUCT
   T : ARRAY  [0 .. 31 ] OF UDT 1010;
  END_STRUCT ;	
BEGIN
END_DATA_BLOCK

